MoveL RelTool (p1,5.500000,12.500000,6.000000,\Rx:=0.000000,\Ry:=0.000000),vel1,zoneval,Extruder\WObj:=Workobject_1;
MoveL RelTool (p1,3.000000,12.500000,6.000000,\Rx:=0.000000,\Ry:=0.000000),vel1,zoneval,Extruder\WObj:=Workobject_1;
MoveL RelTool (p1,5.000000,13.000000,6.000000,\Rx:=0.000000,\Ry:=-0.000000),vel1,zoneval,Extruder\WObj:=Workobject_1;
MoveL RelTool (p1,7.500000,13.000000,6.000000,\Rx:=0.000000,\Ry:=-0.000000),vel1,zoneval,Extruder\WObj:=Workobject_1;
MoveL RelTool (p1,10.000000,13.000000,6.000000,\Rx:=0.000000,\Ry:=-0.000000),vel1,zoneval,Extruder\WObj:=Workobject_1;
MoveL RelTool (p1,12.500000,13.000000,6.000000,\Rx:=0.000000,\Ry:=-0.000000),vel1,zoneval,Extruder\WObj:=Workobject_1;
MoveL RelTool (p1,15.000000,13.000000,6.000000,\Rx:=0.000000,\Ry:=-0.000000),vel1,zoneval,Extruder\WObj:=Workobject_1;
MoveL RelTool (p1,17.500000,13.000000,6.049338,\Rx:=0.000000,\Ry:=-1.971515),vel1,zoneval,Extruder\WObj:=Workobject_1;
MoveL RelTool (p1,20.000000,13.000000,6.980750,\Rx:=0.000000,\Ry:=-8.490094),vel1,zoneval,Extruder\WObj:=Workobject_1;
MoveL RelTool (p1,22.500000,13.000000,9.643620,\Rx:=0.000000,\Ry:=-9.749586),vel1,zoneval,Extruder\WObj:=Workobject_1;
MoveL RelTool (p1,25.000000,13.000000,11.616136,\Rx:=0.000000,\Ry:=-6.984613),vel1,zoneval,Extruder\WObj:=Workobject_1;
MoveL RelTool (p1,27.500000,13.000000,12.963548,\Rx:=0.000000,\Ry:=-5.267415),vel1,zoneval,Extruder\WObj:=Workobject_1;
MoveL RelTool (p1,30.000000,13.000000,13.961706,\Rx:=0.000000,\Ry:=-4.044321),vel1,zoneval,Extruder\WObj:=Workobject_1;
MoveL RelTool (p1,32.500000,13.000000,14.718653,\Rx:=0.000000,\Ry:=-3.050426),vel1,zoneval,Extruder\WObj:=Workobject_1;
MoveL RelTool (p1,35.000000,13.000000,15.272539,\Rx:=0.000000,\Ry:=-2.353997),vel1,zoneval,Extruder\WObj:=Workobject_1;
MoveL RelTool (p1,37.500000,13.000000,15.663580,\Rx:=0.000000,\Ry:=-1.455729),vel1,zoneval,Extruder\WObj:=Workobject_1;
MoveL RelTool (p1,40.000000,13.000000,15.887387,\Rx:=0.000000,\Ry:=-0.888959),vel1,zoneval,Extruder\WObj:=Workobject_1;
MoveL RelTool (p1,42.500000,13.000000,15.992154,\Rx:=0.000000,\Ry:=-0.087941),vel1,zoneval,Extruder\WObj:=Workobject_1;
MoveL RelTool (p1,45.000000,13.000000,15.941430,\Rx:=0.000000,\Ry:=0.668129),vel1,zoneval,Extruder\WObj:=Workobject_1;
MoveL RelTool (p1,47.500000,13.000000,15.759207,\Rx:=0.000000,\Ry:=1.496196),vel1,zoneval,Extruder\WObj:=Workobject_1;
MoveL RelTool (p1,50.000000,13.000000,15.420215,\Rx:=0.000000,\Ry:=2.179974),vel1,zoneval,Extruder\WObj:=Workobject_1;
MoveL RelTool (p1,52.500000,13.000000,14.925537,\Rx:=0.000000,\Ry:=3.343435),vel1,zoneval,Extruder\WObj:=Workobject_1;
MoveL RelTool (p1,55.000000,13.000000,14.234849,\Rx:=0.000000,\Ry:=3.932843),vel1,zoneval,Extruder\WObj:=Workobject_1;
MoveL RelTool (p1,57.500000,13.000000,13.324111,\Rx:=0.000000,\Ry:=5.119588),vel1,zoneval,Extruder\WObj:=Workobject_1;
MoveL RelTool (p1,60.000000,13.000000,12.115065,\Rx:=0.000000,\Ry:=6.738277),vel1,zoneval,Extruder\WObj:=Workobject_1;
MoveL RelTool (p1,62.500000,13.000000,10.412342,\Rx:=0.000000,\Ry:=9.301668),vel1,zoneval,Extruder\WObj:=Workobject_1;
MoveL RelTool (p1,65.000000,13.000000,7.669409,\Rx:=0.000000,\Ry:=9.245058),vel1,zoneval,Extruder\WObj:=Workobject_1;
MoveL RelTool (p1,67.500000,13.000000,6.209438,\Rx:=0.000000,\Ry:=3.081673),vel1,zoneval,Extruder\WObj:=Workobject_1;
MoveL RelTool (p1,70.000000,13.000000,6.000000,\Rx:=0.000000,\Ry:=-0.000000),vel1,zoneval,Extruder\WObj:=Workobject_1;
MoveL RelTool (p1,72.500000,13.000000,6.000000,\Rx:=0.000000,\Ry:=-0.000000),vel1,zoneval,Extruder\WObj:=Workobject_1;
MoveL RelTool (p1,75.000000,13.000000,6.000000,\Rx:=0.000000,\Ry:=-0.000000),vel1,zoneval,Extruder\WObj:=Workobject_1;
MoveL RelTool (p1,77.500000,13.000000,6.000000,\Rx:=0.000000,\Ry:=-0.000000),vel1,zoneval,Extruder\WObj:=Workobject_1;
MoveL RelTool (p1,80.000000,13.000000,6.000000,\Rx:=0.000000,\Ry:=-0.000000),vel1,zoneval,Extruder\WObj:=Workobject_1;
MoveL RelTool (p1,82.500000,13.000000,6.000000,\Rx:=0.000000,\Ry:=-0.000000),vel1,zoneval,Extruder\WObj:=Workobject_1;
MoveL RelTool (p1,80.500000,13.500000,6.000000,\Rx:=0.000000,\Ry:=0.000000),vel1,zoneval,Extruder\WObj:=Workobject_1;
MoveL RelTool (p1,78.000000,13.500000,6.000000,\Rx:=0.000000,\Ry:=0.000000),vel1,zoneval,Extruder\WObj:=Workobject_1;
MoveL RelTool (p1,75.500000,13.500000,6.000000,\Rx:=0.000000,\Ry:=0.000000),vel1,zoneval,Extruder\WObj:=Workobject_1;
MoveL RelTool (p1,73.000000,13.500000,6.000000,\Rx:=0.000000,\Ry:=0.000000),vel1,zoneval,Extruder\WObj:=Workobject_1;
MoveL RelTool (p1,70.500000,13.500000,6.000000,\Rx:=0.000000,\Ry:=0.000000),vel1,zoneval,Extruder\WObj:=Workobject_1;
MoveL RelTool (p1,68.000000,13.500000,6.086002,\Rx:=0.000000,\Ry:=3.081673),vel1,zoneval,Extruder\WObj:=Workobject_1;
MoveL RelTool (p1,65.500000,13.500000,7.225445,\Rx:=0.000000,\Ry:=9.245058),vel1,zoneval,Extruder\WObj:=Workobject_1;
MoveL RelTool (p1,63.000000,13.500000,9.965620,\Rx:=0.000000,\Ry:=9.278495),vel1,zoneval,Extruder\WObj:=Workobject_1;
MoveL RelTool (p1,60.500000,13.500000,11.822412,\Rx:=0.000000,\Ry:=6.739756),vel1,zoneval,Extruder\WObj:=Workobject_1;
MoveL RelTool (p1,58.000000,13.500000,13.112852,\Rx:=0.000000,\Ry:=5.083156),vel1,zoneval,Extruder\WObj:=Workobject_1;
MoveL RelTool (p1,55.500000,13.500000,14.075842,\Rx:=0.000000,\Ry:=3.914347),vel1,zoneval,Extruder\WObj:=Workobject_1;
MoveL RelTool (p1,53.000000,13.500000,14.791119,\Rx:=0.000000,\Ry:=3.343440),vel1,zoneval,Extruder\WObj:=Workobject_1;
MoveL RelTool (p1,50.500000,13.500000,15.333521,\Rx:=0.000000,\Ry:=2.179974),vel1,zoneval,Extruder\WObj:=Workobject_1;
MoveL RelTool (p1,48.000000,13.500000,15.700930,\Rx:=0.000000,\Ry:=1.469323),vel1,zoneval,Extruder\WObj:=Workobject_1;
MoveL RelTool (p1,45.500000,13.500000,15.915465,\Rx:=0.000000,\Ry:=0.668129),vel1,zoneval,Extruder\WObj:=Workobject_1;
MoveL RelTool (p1,43.000000,13.500000,15.995410,\Rx:=0.000000,\Ry:=-0.058203),vel1,zoneval,Extruder\WObj:=Workobject_1;
MoveL RelTool (p1,40.500000,13.500000,15.922527,\Rx:=0.000000,\Ry:=-0.858750),vel1,zoneval,Extruder\WObj:=Workobject_1;
MoveL RelTool (p1,38.000000,13.500000,15.720700,\Rx:=0.000000,\Ry:=-1.431827),vel1,zoneval,Extruder\WObj:=Workobject_1;
MoveL RelTool (p1,35.500000,13.500000,15.365736,\Rx:=0.000000,\Ry:=-2.353997),vel1,zoneval,Extruder\WObj:=Workobject_1;
MoveL RelTool (p1,33.000000,13.500000,14.841013,\Rx:=0.000000,\Ry:=-3.059013),vel1,zoneval,Extruder\WObj:=Workobject_1;
MoveL RelTool (p1,30.500000,13.500000,14.125926,\Rx:=0.000000,\Ry:=-4.044321),vel1,zoneval,Extruder\WObj:=Workobject_1;
MoveL RelTool (p1,28.000000,13.500000,13.182734,\Rx:=0.000000,\Ry:=-5.267415),vel1,zoneval,Extruder\WObj:=Workobject_1;
MoveL RelTool (p1,25.500000,13.500000,11.921360,\Rx:=0.000000,\Ry:=-6.957275),vel1,zoneval,Extruder\WObj:=Workobject_1;
MoveL RelTool (p1,23.000000,13.500000,10.124051,\Rx:=0.000000,\Ry:=-9.725837),vel1,zoneval,Extruder\WObj:=Workobject_1;
MoveL RelTool (p1,20.500000,13.500000,7.374287,\Rx:=0.000000,\Ry:=-8.490094),vel1,zoneval,Extruder\WObj:=Workobject_1;
MoveL RelTool (p1,18.000000,13.500000,6.127384,\Rx:=0.000000,\Ry:=-1.971515),vel1,zoneval,Extruder\WObj:=Workobject_1;
MoveL RelTool (p1,15.500000,13.500000,6.000000,\Rx:=0.000000,\Ry:=0.000000),vel1,zoneval,Extruder\WObj:=Workobject_1;
MoveL RelTool (p1,13.000000,13.500000,6.000000,\Rx:=0.000000,\Ry:=0.000000),vel1,zoneval,Extruder\WObj:=Workobject_1;
MoveL RelTool (p1,10.500000,13.500000,6.000000,\Rx:=0.000000,\Ry:=0.000000),vel1,zoneval,Extruder\WObj:=Workobject_1;
MoveL RelTool (p1,8.000000,13.500000,6.000000,\Rx:=0.000000,\Ry:=0.000000),vel1,zoneval,Extruder\WObj:=Workobject_1;
MoveL RelTool (p1,5.500000,13.500000,6.000000,\Rx:=0.000000,\Ry:=0.000000),vel1,zoneval,Extruder\WObj:=Workobject_1;
MoveL RelTool (p1,3.000000,13.500000,6.000000,\Rx:=0.000000,\Ry:=0.000000),vel1,zoneval,Extruder\WObj:=Workobject_1;
MoveL RelTool (p1,5.000000,14.000000,6.000000,\Rx:=0.000000,\Ry:=-0.000000),vel1,zoneval,Extruder\WObj:=Workobject_1;
MoveL RelTool (p1,7.500000,14.000000,6.000000,\Rx:=0.000000,\Ry:=-0.000000),vel1,zoneval,Extruder\WObj:=Workobject_1;
MoveL RelTool (p1,10.000000,14.000000,6.000000,\Rx:=0.000000,\Ry:=-0.000000),vel1,zoneval,Extruder\WObj:=Workobject_1;
MoveL RelTool (p1,12.500000,14.000000,6.000000,\Rx:=0.000000,\Ry:=-0.000000),vel1,zoneval,Extruder\WObj:=Workobject_1;
MoveL RelTool (p1,15.000000,14.000000,6.000000,\Rx:=0.000000,\Ry:=-0.000000),vel1,zoneval,Extruder\WObj:=Workobject_1;
MoveL RelTool (p1,17.500000,14.000000,6.049338,\Rx:=0.000000,\Ry:=-1.971515),vel1,zoneval,Extruder\WObj:=Workobject_1;
MoveL RelTool (p1,20.000000,14.000000,6.980750,\Rx:=0.000000,\Ry:=-8.490094),vel1,zoneval,Extruder\WObj:=Workobject_1;
MoveL RelTool (p1,22.500000,14.000000,9.646646,\Rx:=0.000000,\Ry:=-9.702002),vel1,zoneval,Extruder\WObj:=Workobject_1;
MoveL RelTool (p1,25.000000,14.000000,11.618390,\Rx:=0.000000,\Ry:=-6.929866),vel1,zoneval,Extruder\WObj:=Workobject_1;
MoveL RelTool (p1,27.500000,14.000000,12.962881,\Rx:=0.000000,\Ry:=-5.267415),vel1,zoneval,Extruder\WObj:=Workobject_1;
MoveL RelTool (p1,30.000000,14.000000,13.961372,\Rx:=0.000000,\Ry:=-4.044321),vel1,zoneval,Extruder\WObj:=Workobject_1;
MoveL RelTool (p1,32.500000,14.000000,14.718387,\Rx:=0.000000,\Ry:=-3.067598),vel1,zoneval,Extruder\WObj:=Workobject_1;
MoveL RelTool (p1,35.000000,14.000000,15.271916,\Rx:=0.000000,\Ry:=-2.353997),vel1,zoneval,Extruder\WObj:=Workobject_1;
MoveL RelTool (p1,37.500000,14.000000,15.664889,\Rx:=0.000000,\Ry:=-1.407915),vel1,zoneval,Extruder\WObj:=Workobject_1;
MoveL RelTool (p1,40.000000,14.000000,15.890119,\Rx:=0.000000,\Ry:=-0.828532),vel1,zoneval,Extruder\WObj:=Workobject_1;
MoveL RelTool (p1,42.500000,14.000000,15.994096,\Rx:=0.000000,\Ry:=-0.028464),vel1,zoneval,Extruder\WObj:=Workobject_1;
MoveL RelTool (p1,45.000000,14.000000,15.942022,\Rx:=0.000000,\Ry:=0.668129),vel1,zoneval,Extruder\WObj:=Workobject_1;
MoveL RelTool (p1,47.500000,14.000000,15.758568,\Rx:=0.000000,\Ry:=1.442437),vel1,zoneval,Extruder\WObj:=Workobject_1;
MoveL RelTool (p1,50.000000,14.000000,15.419734,\Rx:=0.000000,\Ry:=2.179974),vel1,zoneval,Extruder\WObj:=Workobject_1;
MoveL RelTool (p1,52.500000,14.000000,14.925501,\Rx:=0.000000,\Ry:=3.287338),vel1,zoneval,Extruder\WObj:=Workobject_1;
MoveL RelTool (p1,55.000000,14.000000,14.234333,\Rx:=0.000000,\Ry:=3.895833),vel1,zoneval,Extruder\WObj:=Workobject_1;
MoveL RelTool (p1,57.500000,14.000000,13.323479,\Rx:=0.000000,\Ry:=5.046636),vel1,zoneval,Extruder\WObj:=Workobject_1;
MoveL RelTool (p1,60.000000,14.000000,12.114788,\Rx:=0.000000,\Ry:=6.741235),vel1,zoneval,Extruder\WObj:=Workobject_1;
MoveL RelTool (p1,62.500000,14.000000,10.411534,\Rx:=0.000000,\Ry:=9.255247),vel1,zoneval,Extruder\WObj:=Workobject_1;
MoveL RelTool (p1,65.000000,14.000000,7.669409,\Rx:=0.000000,\Ry:=9.245058),vel1,zoneval,Extruder\WObj:=Workobject_1;
MoveL RelTool (p1,67.500000,14.000000,6.209438,\Rx:=0.000000,\Ry:=3.081673),vel1,zoneval,Extruder\WObj:=Workobject_1;
MoveL RelTool (p1,70.000000,14.000000,6.000000,\Rx:=0.000000,\Ry:=-0.000000),vel1,zoneval,Extruder\WObj:=Workobject_1;
MoveL RelTool (p1,72.500000,14.000000,6.000000,\Rx:=0.000000,\Ry:=-0.000000),vel1,zoneval,Extruder\WObj:=Workobject_1;
MoveL RelTool (p1,75.000000,14.000000,6.000000,\Rx:=0.000000,\Ry:=-0.000000),vel1,zoneval,Extruder\WObj:=Workobject_1;
MoveL RelTool (p1,77.500000,14.000000,6.000000,\Rx:=0.000000,\Ry:=-0.000000),vel1,zoneval,Extruder\WObj:=Workobject_1;
MoveL RelTool (p1,80.000000,14.000000,6.000000,\Rx:=0.000000,\Ry:=-0.000000),vel1,zoneval,Extruder\WObj:=Workobject_1;
MoveL RelTool (p1,82.500000,14.000000,6.000000,\Rx:=0.000000,\Ry:=-0.000000),vel1,zoneval,Extruder\WObj:=Workobject_1;
MoveL RelTool (p1,80.500000,14.500000,6.000000,\Rx:=0.000000,\Ry:=0.000000),vel1,zoneval,Extruder\WObj:=Workobject_1;
MoveL RelTool (p1,78.000000,14.500000,6.000000,\Rx:=0.000000,\Ry:=0.000000),vel1,zoneval,Extruder\WObj:=Workobject_1;
MoveL RelTool (p1,75.500000,14.500000,6.000000,\Rx:=0.000000,\Ry:=0.000000),vel1,zoneval,Extruder\WObj:=Workobject_1;
MoveL RelTool (p1,73.000000,14.500000,6.000000,\Rx:=0.000000,\Ry:=0.000000),vel1,zoneval,Extruder\WObj:=Workobject_1;
MoveL RelTool (p1,70.500000,14.500000,6.000000,\Rx:=0.000000,\Ry:=0.000000),vel1,zoneval,Extruder\WObj:=Workobject_1;
MoveL RelTool (p1,68.000000,14.500000,6.086002,\Rx:=0.000000,\Ry:=3.081673),vel1,zoneval,Extruder\WObj:=Workobject_1;
MoveL RelTool (p1,65.500000,14.500000,7.225445,\Rx:=0.000000,\Ry:=9.245058),vel1,zoneval,Extruder\WObj:=Workobject_1;
MoveL RelTool (p1,63.000000,14.500000,9.968088,\Rx:=0.000000,\Ry:=9.231924),vel1,zoneval,Extruder\WObj:=Workobject_1;
MoveL RelTool (p1,60.500000,14.500000,11.821979,\Rx:=0.000000,\Ry:=6.742713),vel1,zoneval,Extruder\WObj:=Workobject_1;
MoveL RelTool (p1,58.000000,14.500000,13.115420,\Rx:=0.000000,\Ry:=5.013820),vel1,zoneval,Extruder\WObj:=Workobject_1;
MoveL RelTool (p1,55.500000,14.500000,14.076926,\Rx:=0.000000,\Ry:=3.877303),vel1,zoneval,Extruder\WObj:=Workobject_1;
MoveL RelTool (p1,53.000000,14.500000,14.795076,\Rx:=0.000000,\Ry:=3.248438),vel1,zoneval,Extruder\WObj:=Workobject_1;
MoveL RelTool (p1,50.500000,14.500000,15.333041,\Rx:=0.000000,\Ry:=2.179974),vel1,zoneval,Extruder\WObj:=Workobject_1;
MoveL RelTool (p1,48.000000,14.500000,15.702430,\Rx:=0.000000,\Ry:=1.415537),vel1,zoneval,Extruder\WObj:=Workobject_1;
MoveL RelTool (p1,45.500000,14.500000,15.916057,\Rx:=0.000000,\Ry:=0.668129),vel1,zoneval,Extruder\WObj:=Workobject_1;
MoveL RelTool (p1,43.000000,14.500000,15.995016,\Rx:=0.000000,\Ry:=0.001275),vel1,zoneval,Extruder\WObj:=Workobject_1;
MoveL RelTool (p1,40.500000,14.500000,15.923861,\Rx:=0.000000,\Ry:=-0.823311),vel1,zoneval,Extruder\WObj:=Workobject_1;
MoveL RelTool (p1,38.000000,14.500000,15.720108,\Rx:=0.000000,\Ry:=-1.383993),vel1,zoneval,Extruder\WObj:=Workobject_1;
MoveL RelTool (p1,35.500000,14.500000,15.365113,\Rx:=0.000000,\Ry:=-2.353997),vel1,zoneval,Extruder\WObj:=Workobject_1;
MoveL RelTool (p1,33.000000,14.500000,14.841462,\Rx:=0.000000,\Ry:=-3.076179),vel1,zoneval,Extruder\WObj:=Workobject_1;
MoveL RelTool (p1,30.500000,14.500000,14.125592,\Rx:=0.000000,\Ry:=-4.044321),vel1,zoneval,Extruder\WObj:=Workobject_1;
MoveL RelTool (p1,28.000000,14.500000,13.182067,\Rx:=0.000000,\Ry:=-5.267415),vel1,zoneval,Extruder\WObj:=Workobject_1;
MoveL RelTool (p1,25.500000,14.500000,11.920669,\Rx:=0.000000,\Ry:=-6.904626),vel1,zoneval,Extruder\WObj:=Workobject_1;
MoveL RelTool (p1,23.000000,14.500000,10.123494,\Rx:=0.000000,\Ry:=-9.678082),vel1,zoneval,Extruder\WObj:=Workobject_1;
MoveL RelTool (p1,20.500000,14.500000,7.374287,\Rx:=0.000000,\Ry:=-8.490094),vel1,zoneval,Extruder\WObj:=Workobject_1;
MoveL RelTool (p1,18.000000,14.500000,6.127384,\Rx:=0.000000,\Ry:=-1.971515),vel1,zoneval,Extruder\WObj:=Workobject_1;
MoveL RelTool (p1,15.500000,14.500000,6.000000,\Rx:=0.000000,\Ry:=0.000000),vel1,zoneval,Extruder\WObj:=Workobject_1;
MoveL RelTool (p1,13.000000,14.500000,6.000000,\Rx:=0.000000,\Ry:=0.000000),vel1,zoneval,Extruder\WObj:=Workobject_1;
MoveL RelTool (p1,10.500000,14.500000,6.000000,\Rx:=0.000000,\Ry:=0.000000),vel1,zoneval,Extruder\WObj:=Workobject_1;
MoveL RelTool (p1,8.000000,14.500000,6.000000,\Rx:=0.000000,\Ry:=0.000000),vel1,zoneval,Extruder\WObj:=Workobject_1;
MoveL RelTool (p1,5.500000,14.500000,6.000000,\Rx:=0.000000,\Ry:=0.000000),vel1,zoneval,Extruder\WObj:=Workobject_1;
MoveL RelTool (p1,3.000000,14.500000,6.000000,\Rx:=0.000000,\Ry:=0.000000),vel1,zoneval,Extruder\WObj:=Workobject_1;
MoveL RelTool (p1,5.000000,15.000000,6.000000,\Rx:=0.000000,\Ry:=-0.000000),vel1,zoneval,Extruder\WObj:=Workobject_1;
MoveL RelTool (p1,7.500000,15.000000,6.000000,\Rx:=0.000000,\Ry:=-0.000000),vel1,zoneval,Extruder\WObj:=Workobject_1;
MoveL RelTool (p1,10.000000,15.000000,6.000000,\Rx:=0.000000,\Ry:=-0.000000),vel1,zoneval,Extruder\WObj:=Workobject_1;
MoveL RelTool (p1,12.500000,15.000000,6.000000,\Rx:=0.000000,\Ry:=-0.000000),vel1,zoneval,Extruder\WObj:=Workobject_1;
MoveL RelTool (p1,15.000000,15.000000,6.000000,\Rx:=0.000000,\Ry:=-0.000000),vel1,zoneval,Extruder\WObj:=Workobject_1;
MoveL RelTool (p1,17.500000,15.000000,6.049338,\Rx:=0.000000,\Ry:=-1.971515),vel1,zoneval,Extruder\WObj:=Workobject_1;
MoveL RelTool (p1,20.000000,15.000000,6.980750,\Rx:=0.000000,\Ry:=-8.490094),vel1,zoneval,Extruder\WObj:=Workobject_1;
MoveL RelTool (p1,22.500000,15.000000,9.649672,\Rx:=0.000000,\Ry:=-9.654076),vel1,zoneval,Extruder\WObj:=Workobject_1;
MoveL RelTool (p1,25.000000,15.000000,11.619515,\Rx:=0.000000,\Ry:=-6.895951),vel1,zoneval,Extruder\WObj:=Workobject_1;
MoveL RelTool (p1,27.500000,15.000000,12.962213,\Rx:=0.000000,\Ry:=-5.267415),vel1,zoneval,Extruder\WObj:=Workobject_1;
MoveL RelTool (p1,30.000000,15.000000,13.961039,\Rx:=0.000000,\Ry:=-4.044321),vel1,zoneval,Extruder\WObj:=Workobject_1;
MoveL RelTool (p1,32.500000,15.000000,14.718121,\Rx:=0.000000,\Ry:=-3.084758),vel1,zoneval,Extruder\WObj:=Workobject_1;
MoveL RelTool (p1,35.000000,15.000000,15.271293,\Rx:=0.000000,\Ry:=-2.353997),vel1,zoneval,Extruder\WObj:=Workobject_1;
MoveL RelTool (p1,37.500000,15.000000,15.666198,\Rx:=0.000000,\Ry:=-1.360061),vel1,zoneval,Extruder\WObj:=Workobject_1;
MoveL RelTool (p1,40.000000,15.000000,15.892850,\Rx:=0.000000,\Ry:=-0.823311),vel1,zoneval,Extruder\WObj:=Workobject_1;
MoveL RelTool (p1,42.500000,15.000000,15.995638,\Rx:=0.000000,\Ry:=0.020861),vel1,zoneval,Extruder\WObj:=Workobject_1;
MoveL RelTool (p1,45.000000,15.000000,15.942614,\Rx:=0.000000,\Ry:=0.668129),vel1,zoneval,Extruder\WObj:=Workobject_1;
MoveL RelTool (p1,47.500000,15.000000,15.757929,\Rx:=0.000000,\Ry:=1.392190),vel1,zoneval,Extruder\WObj:=Workobject_1;
MoveL RelTool (p1,50.000000,15.000000,15.419254,\Rx:=0.000000,\Ry:=2.179974),vel1,zoneval,Extruder\WObj:=Workobject_1;
MoveL RelTool (p1,52.500000,15.000000,14.925466,\Rx:=0.000000,\Ry:=3.209475),vel1,zoneval,Extruder\WObj:=Workobject_1;
MoveL RelTool (p1,55.000000,15.000000,14.233818,\Rx:=0.000000,\Ry:=3.858755),vel1,zoneval,Extruder\WObj:=Workobject_1;
MoveL RelTool (p1,57.500000,15.000000,13.322847,\Rx:=0.000000,\Ry:=5.013820),vel1,zoneval,Extruder\WObj:=Workobject_1;
MoveL RelTool (p1,60.000000,15.000000,12.114512,\Rx:=0.000000,\Ry:=6.744192),vel1,zoneval,Extruder\WObj:=Workobject_1;
MoveL RelTool (p1,62.500000,15.000000,10.410726,\Rx:=0.000000,\Ry:=9.208524),vel1,zoneval,Extruder\WObj:=Workobject_1;
MoveL RelTool (p1,65.000000,15.000000,7.669409,\Rx:=0.000000,\Ry:=9.245058),vel1,zoneval,Extruder\WObj:=Workobject_1;
MoveL RelTool (p1,67.500000,15.000000,6.209438,\Rx:=0.000000,\Ry:=3.081673),vel1,zoneval,Extruder\WObj:=Workobject_1;
MoveL RelTool (p1,70.000000,15.000000,6.000000,\Rx:=0.000000,\Ry:=-0.000000),vel1,zoneval,Extruder\WObj:=Workobject_1;
MoveL RelTool (p1,72.500000,15.000000,6.000000,\Rx:=0.000000,\Ry:=-0.000000),vel1,zoneval,Extruder\WObj:=Workobject_1;
MoveL RelTool (p1,75.000000,15.000000,6.000000,\Rx:=0.000000,\Ry:=-0.000000),vel1,zoneval,Extruder\WObj:=Workobject_1;
MoveL RelTool (p1,77.500000,15.000000,6.000000,\Rx:=0.000000,\Ry:=-0.000000),vel1,zoneval,Extruder\WObj:=Workobject_1;
MoveL RelTool (p1,80.000000,15.000000,6.000000,\Rx:=0.000000,\Ry:=-0.000000),vel1,zoneval,Extruder\WObj:=Workobject_1;
MoveL RelTool (p1,82.500000,15.000000,6.000000,\Rx:=0.000000,\Ry:=-0.000000),vel1,zoneval,Extruder\WObj:=Workobject_1;
MoveL RelTool (p1,80.500000,15.500000,6.000000,\Rx:=0.000000,\Ry:=0.000000),vel1,zoneval,Extruder\WObj:=Workobject_1;
MoveL RelTool (p1,78.000000,15.500000,6.000000,\Rx:=0.000000,\Ry:=0.000000),vel1,zoneval,Extruder\WObj:=Workobject_1;
MoveL RelTool (p1,75.500000,15.500000,6.000000,\Rx:=0.000000,\Ry:=0.000000),vel1,zoneval,Extruder\WObj:=Workobject_1;
MoveL RelTool (p1,73.000000,15.500000,6.000000,\Rx:=0.000000,\Ry:=0.000000),vel1,zoneval,Extruder\WObj:=Workobject_1;
MoveL RelTool (p1,70.500000,15.500000,6.000000,\Rx:=0.000000,\Ry:=0.000000),vel1,zoneval,Extruder\WObj:=Workobject_1;
MoveL RelTool (p1,68.000000,15.500000,6.086002,\Rx:=0.000000,\Ry:=3.081673),vel1,zoneval,Extruder\WObj:=Workobject_1;
MoveL RelTool (p1,65.500000,15.500000,7.225445,\Rx:=0.000000,\Ry:=9.245058),vel1,zoneval,Extruder\WObj:=Workobject_1;
MoveL RelTool (p1,63.000000,15.500000,9.970555,\Rx:=0.000000,\Ry:=9.185048),vel1,zoneval,Extruder\WObj:=Workobject_1;
MoveL RelTool (p1,60.500000,15.500000,11.821547,\Rx:=0.000000,\Ry:=6.745670),vel1,zoneval,Extruder\WObj:=Workobject_1;
MoveL RelTool (p1,58.000000,15.500000,13.114788,\Rx:=0.000000,\Ry:=5.013820),vel1,zoneval,Extruder\WObj:=Workobject_1;
MoveL RelTool (p1,55.500000,15.500000,14.078010,\Rx:=0.000000,\Ry:=3.840191),vel1,zoneval,Extruder\WObj:=Workobject_1;
MoveL RelTool (p1,53.000000,15.500000,14.798306,\Rx:=0.000000,\Ry:=3.170451),vel1,zoneval,Extruder\WObj:=Workobject_1;
MoveL RelTool (p1,50.500000,15.500000,15.332561,\Rx:=0.000000,\Ry:=2.179974),vel1,zoneval,Extruder\WObj:=Workobject_1;
MoveL RelTool (p1,48.000000,15.500000,15.703432,\Rx:=0.000000,\Ry:=1.374237),vel1,zoneval,Extruder\WObj:=Workobject_1;
MoveL RelTool (p1,45.500000,15.500000,15.916648,\Rx:=0.000000,\Ry:=0.668129),vel1,zoneval,Extruder\WObj:=Workobject_1;
MoveL RelTool (p1,43.000000,15.500000,15.994622,\Rx:=0.000000,\Ry:=0.023524),vel1,zoneval,Extruder\WObj:=Workobject_1;
MoveL RelTool (p1,40.500000,15.500000,15.926593,\Rx:=0.000000,\Ry:=-0.823311),vel1,zoneval,Extruder\WObj:=Workobject_1;
MoveL RelTool (p1,38.000000,15.500000,15.719515,\Rx:=0.000000,\Ry:=-1.336120),vel1,zoneval,Extruder\WObj:=Workobject_1;
MoveL RelTool (p1,35.500000,15.500000,15.364490,\Rx:=0.000000,\Ry:=-2.353997),vel1,zoneval,Extruder\WObj:=Workobject_1;
MoveL RelTool (p1,33.000000,15.500000,14.841911,\Rx:=0.000000,\Ry:=-3.093334),vel1,zoneval,Extruder\WObj:=Workobject_1;
MoveL RelTool (p1,30.500000,15.500000,14.125258,\Rx:=0.000000,\Ry:=-4.044321),vel1,zoneval,Extruder\WObj:=Workobject_1;
MoveL RelTool (p1,28.000000,15.500000,13.181399,\Rx:=0.000000,\Ry:=-5.267415),vel1,zoneval,Extruder\WObj:=Workobject_1;
MoveL RelTool (p1,25.500000,15.500000,11.919977,\Rx:=0.000000,\Ry:=-6.887269),vel1,zoneval,Extruder\WObj:=Workobject_1;
MoveL RelTool (p1,23.000000,15.500000,10.122937,\Rx:=0.000000,\Ry:=-9.629984),vel1,zoneval,Extruder\WObj:=Workobject_1;
MoveL RelTool (p1,20.500000,15.500000,7.374287,\Rx:=0.000000,\Ry:=-8.490094),vel1,zoneval,Extruder\WObj:=Workobject_1;
MoveL RelTool (p1,18.000000,15.500000,6.127384,\Rx:=0.000000,\Ry:=-1.971515),vel1,zoneval,Extruder\WObj:=Workobject_1;
MoveL RelTool (p1,15.500000,15.500000,6.000000,\Rx:=0.000000,\Ry:=0.000000),vel1,zoneval,Extruder\WObj:=Workobject_1;
MoveL RelTool (p1,13.000000,15.500000,6.000000,\Rx:=0.000000,\Ry:=0.000000),vel1,zoneval,Extruder\WObj:=Workobject_1;
MoveL RelTool (p1,10.500000,15.500000,6.000000,\Rx:=0.000000,\Ry:=0.000000),vel1,zoneval,Extruder\WObj:=Workobject_1;
MoveL RelTool (p1,8.000000,15.500000,6.000000,\Rx:=0.000000,\Ry:=0.000000),vel1,zoneval,Extruder\WObj:=Workobject_1;
MoveL RelTool (p1,5.500000,15.500000,6.000000,\Rx:=0.000000,\Ry:=0.000000),vel1,zoneval,Extruder\WObj:=Workobject_1;
MoveL RelTool (p1,3.000000,15.500000,6.000000,\Rx:=0.000000,\Ry:=0.000000),vel1,zoneval,Extruder\WObj:=Workobject_1;
MoveL RelTool (p1,5.000000,16.000000,6.000000,\Rx:=0.000000,\Ry:=-0.000000),vel1,zoneval,Extruder\WObj:=Workobject_1;
MoveL RelTool (p1,7.500000,16.000000,6.000000,\Rx:=0.000000,\Ry:=-0.000000),vel1,zoneval,Extruder\WObj:=Workobject_1;
MoveL RelTool (p1,10.000000,16.000000,6.000000,\Rx:=0.000000,\Ry:=-0.000000),vel1,zoneval,Extruder\WObj:=Workobject_1;
MoveL RelTool (p1,12.500000,16.000000,6.000000,\Rx:=0.000000,\Ry:=-0.000000),vel1,zoneval,Extruder\WObj:=Workobject_1;
MoveL RelTool (p1,15.000000,16.000000,6.000000,\Rx:=0.000000,\Ry:=-0.000000),vel1,zoneval,Extruder\WObj:=Workobject_1;
MoveL RelTool (p1,17.500000,16.000000,6.049338,\Rx:=0.000000,\Ry:=-1.971515),vel1,zoneval,Extruder\WObj:=Workobject_1;
MoveL RelTool (p1,20.000000,16.000000,6.980750,\Rx:=0.000000,\Ry:=-8.490094),vel1,zoneval,Extruder\WObj:=Workobject_1;
MoveL RelTool (p1,22.500000,16.000000,9.652698,\Rx:=0.000000,\Ry:=-9.605805),vel1,zoneval,Extruder\WObj:=Workobject_1;
MoveL RelTool (p1,25.000000,16.000000,11.619752,\Rx:=0.000000,\Ry:=-6.878580),vel1,zoneval,Extruder\WObj:=Workobject_1;
MoveL RelTool (p1,27.500000,16.000000,12.961545,\Rx:=0.000000,\Ry:=-5.267415),vel1,zoneval,Extruder\WObj:=Workobject_1;
MoveL RelTool (p1,30.000000,16.000000,13.960705,\Rx:=0.000000,\Ry:=-4.044321),vel1,zoneval,Extruder\WObj:=Workobject_1;
MoveL RelTool (p1,32.500000,16.000000,14.717855,\Rx:=0.000000,\Ry:=-3.101906),vel1,zoneval,Extruder\WObj:=Workobject_1;
MoveL RelTool (p1,35.000000,16.000000,15.270669,\Rx:=0.000000,\Ry:=-2.353997),vel1,zoneval,Extruder\WObj:=Workobject_1;
MoveL RelTool (p1,37.500000,16.000000,15.667148,\Rx:=0.000000,\Ry:=-1.321199),vel1,zoneval,Extruder\WObj:=Workobject_1;
MoveL RelTool (p1,40.000000,16.000000,15.895582,\Rx:=0.000000,\Ry:=-0.823311),vel1,zoneval,Extruder\WObj:=Workobject_1;
MoveL RelTool (p1,42.500000,16.000000,15.995453,\Rx:=0.000000,\Ry:=0.026186),vel1,zoneval,Extruder\WObj:=Workobject_1;
MoveL RelTool (p1,45.000000,16.000000,15.943206,\Rx:=0.000000,\Ry:=0.668129),vel1,zoneval,Extruder\WObj:=Workobject_1;
MoveL RelTool (p1,47.500000,16.000000,15.757289,\Rx:=0.000000,\Ry:=1.356278),vel1,zoneval,Extruder\WObj:=Workobject_1;
MoveL RelTool (p1,50.000000,16.000000,15.418774,\Rx:=0.000000,\Ry:=2.179974),vel1,zoneval,Extruder\WObj:=Workobject_1;
MoveL RelTool (p1,52.500000,16.000000,14.925430,\Rx:=0.000000,\Ry:=3.131366),vel1,zoneval,Extruder\WObj:=Workobject_1;
MoveL RelTool (p1,55.000000,16.000000,14.233302,\Rx:=0.000000,\Ry:=3.821610),vel1,zoneval,Extruder\WObj:=Workobject_1;
MoveL RelTool (p1,57.500000,16.000000,13.322215,\Rx:=0.000000,\Ry:=5.013820),vel1,zoneval,Extruder\WObj:=Workobject_1;
MoveL RelTool (p1,60.000000,16.000000,12.114235,\Rx:=0.000000,\Ry:=6.747148),vel1,zoneval,Extruder\WObj:=Workobject_1;
MoveL RelTool (p1,62.500000,16.000000,10.409918,\Rx:=0.000000,\Ry:=9.161496),vel1,zoneval,Extruder\WObj:=Workobject_1;
MoveL RelTool (p1,65.000000,16.000000,7.669409,\Rx:=0.000000,\Ry:=9.245058),vel1,zoneval,Extruder\WObj:=Workobject_1;
MoveL RelTool (p1,67.500000,16.000000,6.209438,\Rx:=0.000000,\Ry:=3.081673),vel1,zoneval,Extruder\WObj:=Workobject_1;
MoveL RelTool (p1,70.000000,16.000000,6.000000,\Rx:=0.000000,\Ry:=-0.000000),vel1,zoneval,Extruder\WObj:=Workobject_1;
MoveL RelTool (p1,72.500000,16.000000,6.000000,\Rx:=0.000000,\Ry:=-0.000000),vel1,zoneval,Extruder\WObj:=Workobject_1;
MoveL RelTool (p1,75.000000,16.000000,6.000000,\Rx:=0.000000,\Ry:=-0.000000),vel1,zoneval,Extruder\WObj:=Workobject_1;
MoveL RelTool (p1,77.500000,16.000000,6.000000,\Rx:=0.000000,\Ry:=-0.000000),vel1,zoneval,Extruder\WObj:=Workobject_1;
MoveL RelTool (p1,80.000000,16.000000,6.000000,\Rx:=0.000000,\Ry:=-0.000000),vel1,zoneval,Extruder\WObj:=Workobject_1;
MoveL RelTool (p1,82.500000,16.000000,6.000000,\Rx:=0.000000,\Ry:=-0.000000),vel1,zoneval,Extruder\WObj:=Workobject_1;



MoveL RelTool (p1,82.500000,16.000000,70.000000,\Rx:=0.000000,\Ry:=-0.000000),vel1,zoneval,Extruder\WObj:=Workobject_1;



MoveL RelTool (p1,3.000000,3.000000,70.000000,\Rx:=0.000000,\Ry:=-0.000000),vel1,zoneval,Extruder\WObj:=Workobject_1;




MoveL RelTool (p1,3.000000,3.000000,6.500000,\Rx:=0.000000,\Ry:=0.000000),vel1,z0,Extruder\WObj:=Workobject_1;
MoveL RelTool (p1,16.889791,3.000000,6.500000,\Rx:=0.000000,\Ry:=0.000000),vel1,z0,Extruder\WObj:=Workobject_1;
MoveL RelTool (p1,17.693081,3.000000,6.564949,\Rx:=0.000000,\Ry:=0.000000),vel1,z0,Extruder\WObj:=Workobject_1;
MoveL RelTool (p1,18.475496,3.000000,6.758109,\Rx:=0.000000,\Ry:=0.000000),vel1,z0,Extruder\WObj:=Workobject_1;
MoveL RelTool (p1,19.216721,3.000000,7.074461,\Rx:=0.000000,\Ry:=0.000000),vel1,z0,Extruder\WObj:=Workobject_1;
MoveL RelTool (p1,19.897491,3.000000,7.505786,\Rx:=0.000000,\Ry:=0.000000),vel1,z0,Extruder\WObj:=Workobject_1;
MoveL RelTool (p1,20.500122,3.000000,8.040880,\Rx:=0.000000,\Ry:=0.000000),vel1,z0,Extruder\WObj:=Workobject_1;
MoveL RelTool (p1,21.008959,3.000000,8.665841,\Rx:=0.000000,\Ry:=0.000000),vel1,z0,Extruder\WObj:=Workobject_1;
MoveL RelTool (p1,21.655001,3.000000,9.492284,\Rx:=0.000000,\Ry:=0.000000),vel1,z0,Extruder\WObj:=Workobject_1;
MoveL RelTool (p1,22.745361,3.000000,10.576250,\Rx:=0.000000,\Ry:=0.000000),vel1,z0,Extruder\WObj:=Workobject_1;
MoveL RelTool (p1,24.141754,3.000000,11.657135,\Rx:=0.000000,\Ry:=0.000000),vel1,z0,Extruder\WObj:=Workobject_1;
MoveL RelTool (p1,25.864042,3.000000,12.709541,\Rx:=0.000000,\Ry:=0.000000),vel1,z0,Extruder\WObj:=Workobject_1;
MoveL RelTool (p1,27.915775,3.000000,13.697697,\Rx:=0.000000,\Ry:=0.000000),vel1,z0,Extruder\WObj:=Workobject_1;
MoveL RelTool (p1,30.224897,3.000000,14.569467,\Rx:=0.000000,\Ry:=0.000000),vel1,z0,Extruder\WObj:=Workobject_1;
MoveL RelTool (p1,32.769985,3.000000,15.305704,\Rx:=0.000000,\Ry:=0.000000),vel1,z0,Extruder\WObj:=Workobject_1;
MoveL RelTool (p1,35.546967,3.000000,15.885172,\Rx:=0.000000,\Ry:=0.000000),vel1,z0,Extruder\WObj:=Workobject_1;
MoveL RelTool (p1,38.467556,3.000000,16.278698,\Rx:=0.000000,\Ry:=0.000000),vel1,z0,Extruder\WObj:=Workobject_1;
MoveL RelTool (p1,41.456455,3.000000,16.476196,\Rx:=0.000000,\Ry:=0.000000),vel1,z0,Extruder\WObj:=Workobject_1;
MoveL RelTool (p1,44.466969,3.000000,16.473138,\Rx:=0.000000,\Ry:=0.000000),vel1,z0,Extruder\WObj:=Workobject_1;
MoveL RelTool (p1,47.447681,3.000000,16.270333,\Rx:=0.000000,\Ry:=0.000000),vel1,z0,Extruder\WObj:=Workobject_1;
MoveL RelTool (p1,50.292072,3.000000,15.884033,\Rx:=0.000000,\Ry:=0.000000),vel1,z0,Extruder\WObj:=Workobject_1;
MoveL RelTool (p1,52.986897,3.000000,15.324379,\Rx:=0.000000,\Ry:=0.000000),vel1,z0,Extruder\WObj:=Workobject_1;
MoveL RelTool (p1,55.503719,3.000000,14.603756,\Rx:=0.000000,\Ry:=0.000000),vel1,z0,Extruder\WObj:=Workobject_1;
MoveL RelTool (p1,57.756004,3.000000,13.765661,\Rx:=0.000000,\Ry:=0.000000),vel1,z0,Extruder\WObj:=Workobject_1;
MoveL RelTool (p1,59.724201,3.000000,12.840277,\Rx:=0.000000,\Ry:=0.000000),vel1,z0,Extruder\WObj:=Workobject_1;
MoveL RelTool (p1,61.421394,3.000000,11.838728,\Rx:=0.000000,\Ry:=0.000000),vel1,z0,Extruder\WObj:=Workobject_1;
MoveL RelTool (p1,62.837132,3.000000,10.789865,\Rx:=0.000000,\Ry:=0.000000),vel1,z0,Extruder\WObj:=Workobject_1;
MoveL RelTool (p1,63.967651,3.000000,9.724504,\Rx:=0.000000,\Ry:=0.000000),vel1,z0,Extruder\WObj:=Workobject_1;
MoveL RelTool (p1,64.823410,3.000000,8.665841,\Rx:=0.000000,\Ry:=0.000000),vel1,z0,Extruder\WObj:=Workobject_1;
MoveL RelTool (p1,65.332253,3.000000,8.040880,\Rx:=0.000000,\Ry:=0.000000),vel1,z0,Extruder\WObj:=Workobject_1;
MoveL RelTool (p1,65.934883,3.000000,7.505786,\Rx:=0.000000,\Ry:=0.000000),vel1,z0,Extruder\WObj:=Workobject_1;
MoveL RelTool (p1,66.615646,3.000000,7.074461,\Rx:=0.000000,\Ry:=0.000000),vel1,z0,Extruder\WObj:=Workobject_1;
MoveL RelTool (p1,67.356880,3.000000,6.758109,\Rx:=0.000000,\Ry:=0.000000),vel1,z0,Extruder\WObj:=Workobject_1;
MoveL RelTool (p1,68.139290,3.000000,6.564949,\Rx:=0.000000,\Ry:=0.000000),vel1,z0,Extruder\WObj:=Workobject_1;
MoveL RelTool (p1,68.942581,3.000000,6.500000,\Rx:=0.000000,\Ry:=0.000000),vel1,z0,Extruder\WObj:=Workobject_1;
MoveL RelTool (p1,82.832375,3.000000,6.500000,\Rx:=0.000000,\Ry:=0.000000),vel1,z0,Extruder\WObj:=Workobject_1;
MoveL RelTool (p1,82.832375,16.000000,6.500000,\Rx:=0.000000,\Ry:=0.000000),vel1,z0,Extruder\WObj:=Workobject_1;
MoveL RelTool (p1,68.942581,16.000000,6.500000,\Rx:=0.000000,\Ry:=0.000000),vel1,z0,Extruder\WObj:=Workobject_1;
MoveL RelTool (p1,68.139290,16.000000,6.564949,\Rx:=0.000000,\Ry:=0.000000),vel1,z0,Extruder\WObj:=Workobject_1;
MoveL RelTool (p1,67.356880,16.000000,6.758109,\Rx:=0.000000,\Ry:=0.000000),vel1,z0,Extruder\WObj:=Workobject_1;
MoveL RelTool (p1,66.615646,16.000000,7.074461,\Rx:=0.000000,\Ry:=0.000000),vel1,z0,Extruder\WObj:=Workobject_1;
MoveL RelTool (p1,65.934883,16.000000,7.505786,\Rx:=0.000000,\Ry:=0.000000),vel1,z0,Extruder\WObj:=Workobject_1;
MoveL RelTool (p1,65.332253,16.000000,8.040880,\Rx:=0.000000,\Ry:=0.000000),vel1,z0,Extruder\WObj:=Workobject_1;
MoveL RelTool (p1,64.823410,16.000000,8.665841,\Rx:=0.000000,\Ry:=0.000000),vel1,z0,Extruder\WObj:=Workobject_1;
MoveL RelTool (p1,64.363686,16.000000,9.273595,\Rx:=0.000000,\Ry:=0.000000),vel1,z0,Extruder\WObj:=Workobject_1;
MoveL RelTool (p1,63.963219,16.000000,9.720532,\Rx:=0.000000,\Ry:=0.000000),vel1,z0,Extruder\WObj:=Workobject_1;
MoveL RelTool (p1,63.821823,16.000000,9.878342,\Rx:=0.000000,\Ry:=0.000000),vel1,z0,Extruder\WObj:=Workobject_1;
MoveL RelTool (p1,63.165062,16.000000,10.507496,\Rx:=0.000000,\Ry:=0.000000),vel1,z0,Extruder\WObj:=Workobject_1;
MoveL RelTool (p1,62.831947,16.000000,10.783607,\Rx:=0.000000,\Ry:=0.000000),vel1,z0,Extruder\WObj:=Workobject_1;
MoveL RelTool (p1,62.416321,16.000000,11.128095,\Rx:=0.000000,\Ry:=0.000000),vel1,z0,Extruder\WObj:=Workobject_1;
MoveL RelTool (p1,61.578415,16.000000,11.733726,\Rx:=0.000000,\Ry:=0.000000),vel1,z0,Extruder\WObj:=Workobject_1;
MoveL RelTool (p1,61.418831,16.000000,11.834675,\Rx:=0.000000,\Ry:=0.000000),vel1,z0,Extruder\WObj:=Workobject_1;
MoveL RelTool (p1,60.616638,16.000000,12.342117,\Rx:=0.000000,\Ry:=0.000000),vel1,z0,Extruder\WObj:=Workobject_1;
MoveL RelTool (p1,59.722591,16.000000,12.837377,\Rx:=0.000000,\Ry:=0.000000),vel1,z0,Extruder\WObj:=Workobject_1;
MoveL RelTool (p1,59.593624,16.000000,12.908818,\Rx:=0.000000,\Ry:=0.000000),vel1,z0,Extruder\WObj:=Workobject_1;
MoveL RelTool (p1,58.474972,16.000000,13.452054,\Rx:=0.000000,\Ry:=0.000000),vel1,z0,Extruder\WObj:=Workobject_1;
MoveL RelTool (p1,57.753036,16.000000,13.758680,\Rx:=0.000000,\Ry:=0.000000),vel1,z0,Extruder\WObj:=Workobject_1;
MoveL RelTool (p1,57.254681,16.000000,13.970348,\Rx:=0.000000,\Ry:=0.000000),vel1,z0,Extruder\WObj:=Workobject_1;
MoveL RelTool (p1,55.907604,16.000000,14.468318,\Rx:=0.000000,\Ry:=0.000000),vel1,z0,Extruder\WObj:=Workobject_1;
MoveL RelTool (p1,55.501736,16.000000,14.597532,\Rx:=0.000000,\Ry:=0.000000),vel1,z0,Extruder\WObj:=Workobject_1;
MoveL RelTool (p1,54.486706,16.000000,14.920681,\Rx:=0.000000,\Ry:=0.000000),vel1,z0,Extruder\WObj:=Workobject_1;
MoveL RelTool (p1,53.019268,16.000000,15.316940,\Rx:=0.000000,\Ry:=0.000000),vel1,z0,Extruder\WObj:=Workobject_1;
MoveL RelTool (p1,52.986862,16.000000,15.324217,\Rx:=0.000000,\Ry:=0.000000),vel1,z0,Extruder\WObj:=Workobject_1;
MoveL RelTool (p1,51.488445,16.000000,15.660700,\Rx:=0.000000,\Ry:=0.000000),vel1,z0,Extruder\WObj:=Workobject_1;
MoveL RelTool (p1,50.290966,16.000000,15.877948,\Rx:=0.000000,\Ry:=0.000000),vel1,z0,Extruder\WObj:=Workobject_1;
MoveL RelTool (p1,49.889133,16.000000,15.950849,\Rx:=0.000000,\Ry:=0.000000),vel1,z0,Extruder\WObj:=Workobject_1;
MoveL RelTool (p1,48.224419,16.000000,16.184232,\Rx:=0.000000,\Ry:=0.000000),vel1,z0,Extruder\WObj:=Workobject_1;
MoveL RelTool (p1,47.446861,16.000000,16.262141,\Rx:=0.000000,\Ry:=0.000000),vel1,z0,Extruder\WObj:=Workobject_1;
MoveL RelTool (p1,46.521641,16.000000,16.354847,\Rx:=0.000000,\Ry:=0.000000),vel1,z0,Extruder\WObj:=Workobject_1;
MoveL RelTool (p1,44.783478,16.000000,16.461150,\Rx:=0.000000,\Ry:=0.000000),vel1,z0,Extruder\WObj:=Workobject_1;
MoveL RelTool (p1,44.466858,16.000000,16.468186,\Rx:=0.000000,\Ry:=0.000000),vel1,z0,Extruder\WObj:=Workobject_1;
MoveL RelTool (p1,43.043808,16.000000,16.499818,\Rx:=0.000000,\Ry:=0.000000),vel1,z0,Extruder\WObj:=Workobject_1;
MoveL RelTool (p1,41.456497,16.000000,16.473560,\Rx:=0.000000,\Ry:=0.000000),vel1,z0,Extruder\WObj:=Workobject_1;
MoveL RelTool (p1,41.303349,16.000000,16.471027,\Rx:=0.000000,\Ry:=0.000000),vel1,z0,Extruder\WObj:=Workobject_1;
MoveL RelTool (p1,39.566307,16.000000,16.374732,\Rx:=0.000000,\Ry:=0.000000),vel1,z0,Extruder\WObj:=Workobject_1;
MoveL RelTool (p1,38.468281,16.000000,16.271000,\Rx:=0.000000,\Ry:=0.000000),vel1,z0,Extruder\WObj:=Workobject_1;
MoveL RelTool (p1,37.849564,16.000000,16.212550,\Rx:=0.000000,\Ry:=0.000000),vel1,z0,Extruder\WObj:=Workobject_1;
MoveL RelTool (p1,36.162739,16.000000,15.985516,\Rx:=0.000000,\Ry:=0.000000),vel1,z0,Extruder\WObj:=Workobject_1;
MoveL RelTool (p1,35.548347,16.000000,15.877330,\Rx:=0.000000,\Ry:=0.000000),vel1,z0,Extruder\WObj:=Workobject_1;
MoveL RelTool (p1,34.531830,16.000000,15.698334,\Rx:=0.000000,\Ry:=0.000000),vel1,z0,Extruder\WObj:=Workobject_1;
MoveL RelTool (p1,32.962124,16.000000,15.353427,\Rx:=0.000000,\Ry:=0.000000),vel1,z0,Extruder\WObj:=Workobject_1;
MoveL RelTool (p1,32.770821,16.000000,15.302555,\Rx:=0.000000,\Ry:=0.000000),vel1,z0,Extruder\WObj:=Workobject_1;
MoveL RelTool (p1,31.457693,16.000000,14.953369,\Rx:=0.000000,\Ry:=0.000000),vel1,z0,Extruder\WObj:=Workobject_1;
MoveL RelTool (p1,30.226080,16.000000,14.565704,\Rx:=0.000000,\Ry:=0.000000),vel1,z0,Extruder\WObj:=Workobject_1;
MoveL RelTool (p1,30.018776,16.000000,14.500453,\Rx:=0.000000,\Ry:=0.000000),vel1,z0,Extruder\WObj:=Workobject_1;
MoveL RelTool (p1,28.659712,16.000000,14.002768,\Rx:=0.000000,\Ry:=0.000000),vel1,z0,Extruder\WObj:=Workobject_1;
MoveL RelTool (p1,27.918875,16.000000,13.690347,\Rx:=0.000000,\Ry:=0.000000),vel1,z0,Extruder\WObj:=Workobject_1;
MoveL RelTool (p1,27.404802,16.000000,13.473557,\Rx:=0.000000,\Ry:=0.000000),vel1,z0,Extruder\WObj:=Workobject_1;
MoveL RelTool (p1,26.235151,16.000000,12.906940,\Rx:=0.000000,\Ry:=0.000000),vel1,z0,Extruder\WObj:=Workobject_1;
MoveL RelTool (p1,25.867798,16.000000,12.702785,\Rx:=0.000000,\Ry:=0.000000),vel1,z0,Extruder\WObj:=Workobject_1;
MoveL RelTool (p1,25.171089,16.000000,12.315596,\Rx:=0.000000,\Ry:=0.000000),vel1,z0,Extruder\WObj:=Workobject_1;
MoveL RelTool (p1,24.206091,16.000000,11.701200,\Rx:=0.000000,\Ry:=0.000000),vel1,z0,Extruder\WObj:=Workobject_1;
MoveL RelTool (p1,24.143076,16.000000,11.655322,\Rx:=0.000000,\Ry:=0.000000),vel1,z0,Extruder\WObj:=Workobject_1;
MoveL RelTool (p1,23.372747,16.000000,11.094489,\Rx:=0.000000,\Ry:=0.000000),vel1,z0,Extruder\WObj:=Workobject_1;
MoveL RelTool (p1,22.748590,16.000000,10.572390,\Rx:=0.000000,\Ry:=0.000000),vel1,z0,Extruder\WObj:=Workobject_1;
MoveL RelTool (p1,22.615110,16.000000,10.460735,\Rx:=0.000000,\Ry:=0.000000),vel1,z0,Extruder\WObj:=Workobject_1;
MoveL RelTool (p1,21.967155,16.000000,9.833263,\Rx:=0.000000,\Ry:=0.000000),vel1,z0,Extruder\WObj:=Workobject_1;
MoveL RelTool (p1,21.661156,16.000000,9.486848,\Rx:=0.000000,\Ry:=0.000000),vel1,z0,Extruder\WObj:=Workobject_1;
MoveL RelTool (p1,21.416798,16.000000,9.210219,\Rx:=0.000000,\Ry:=0.000000),vel1,z0,Extruder\WObj:=Workobject_1;
MoveL RelTool (p1,21.008959,16.000000,8.665841,\Rx:=0.000000,\Ry:=0.000000),vel1,z0,Extruder\WObj:=Workobject_1;
MoveL RelTool (p1,20.500122,16.000000,8.040880,\Rx:=0.000000,\Ry:=0.000000),vel1,z0,Extruder\WObj:=Workobject_1;
MoveL RelTool (p1,19.897491,16.000000,7.505786,\Rx:=0.000000,\Ry:=0.000000),vel1,z0,Extruder\WObj:=Workobject_1;
MoveL RelTool (p1,19.216721,16.000000,7.074461,\Rx:=0.000000,\Ry:=0.000000),vel1,z0,Extruder\WObj:=Workobject_1;
MoveL RelTool (p1,18.475496,16.000000,6.758109,\Rx:=0.000000,\Ry:=0.000000),vel1,z0,Extruder\WObj:=Workobject_1;
MoveL RelTool (p1,17.693081,16.000000,6.564949,\Rx:=0.000000,\Ry:=0.000000),vel1,z0,Extruder\WObj:=Workobject_1;
MoveL RelTool (p1,16.889791,16.000000,6.500000,\Rx:=0.000000,\Ry:=0.000000),vel1,z0,Extruder\WObj:=Workobject_1;
MoveL RelTool (p1,3.000000,16.000000,6.500000,\Rx:=0.000000,\Ry:=0.000000),vel1,z0,Extruder\WObj:=Workobject_1;
MoveL RelTool (p1,3.000000,3.000000,6.500000,\Rx:=0.000000,\Ry:=0.000000),vel1,z0,Extruder\WObj:=Workobject_1;


MoveL RelTool (p1,3.000000,3.000000,6.500000,\Rx:=0.000000,\Ry:=0),vel1,zoneval,Extruder\WObj:=Workobject_1;
MoveL RelTool (p1,5.000000,3.000000,6.500000,\Rx:=0.000000,\Ry:=-0.000000),vel1,zoneval,Extruder\WObj:=Workobject_1;
MoveL RelTool (p1,7.500000,3.000000,6.500000,\Rx:=0.000000,\Ry:=-0.000000),vel1,zoneval,Extruder\WObj:=Workobject_1;
MoveL RelTool (p1,10.000000,3.000000,6.500000,\Rx:=0.000000,\Ry:=-0.000000),vel1,zoneval,Extruder\WObj:=Workobject_1;
MoveL RelTool (p1,12.500000,3.000000,6.500000,\Rx:=0.000000,\Ry:=-0.000000),vel1,zoneval,Extruder\WObj:=Workobject_1;
MoveL RelTool (p1,15.000000,3.000000,6.500000,\Rx:=0.000000,\Ry:=-0.000000),vel1,zoneval,Extruder\WObj:=Workobject_1;
MoveL RelTool (p1,17.500000,3.000000,6.549338,\Rx:=0.000000,\Ry:=-2.301628),vel1,zoneval,Extruder\WObj:=Workobject_1;
MoveL RelTool (p1,20.000000,3.000000,7.596807,\Rx:=0.000000,\Ry:=-9.245074),vel1,zoneval,Extruder\WObj:=Workobject_1;
MoveL RelTool (p1,22.500000,3.000000,10.332328,\Rx:=0.000000,\Ry:=-9.203115),vel1,zoneval,Extruder\WObj:=Workobject_1;
MoveL RelTool (p1,25.000000,3.000000,12.181567,\Rx:=0.000000,\Ry:=-6.983793),vel1,zoneval,Extruder\WObj:=Workobject_1;
MoveL RelTool (p1,27.500000,3.000000,13.497451,\Rx:=0.000000,\Ry:=-5.532306),vel1,zoneval,Extruder\WObj:=Workobject_1;
MoveL RelTool (p1,30.000000,3.000000,14.484560,\Rx:=0.000000,\Ry:=-4.046642),vel1,zoneval,Extruder\WObj:=Workobject_1;
MoveL RelTool (p1,32.500000,3.000000,15.227603,\Rx:=0.000000,\Ry:=-3.145456),vel1,zoneval,Extruder\WObj:=Workobject_1;
MoveL RelTool (p1,35.000000,3.000000,15.771037,\Rx:=0.000000,\Ry:=-2.619262),vel1,zoneval,Extruder\WObj:=Workobject_1;
MoveL RelTool (p1,37.500000,3.000000,16.148328,\Rx:=0.000000,\Ry:=-1.705318),vel1,zoneval,Extruder\WObj:=Workobject_1;
MoveL RelTool (p1,40.000000,3.000000,16.379958,\Rx:=0.000000,\Ry:=-0.840101),vel1,zoneval,Extruder\WObj:=Workobject_1;
MoveL RelTool (p1,42.500000,3.000000,16.475136,\Rx:=0.000000,\Ry:=0.012935),vel1,zoneval,Extruder\WObj:=Workobject_1;
MoveL RelTool (p1,45.000000,3.000000,16.436871,\Rx:=0.000000,\Ry:=0.864966),vel1,zoneval,Extruder\WObj:=Workobject_1;
MoveL RelTool (p1,47.500000,3.000000,16.263228,\Rx:=0.000000,\Ry:=1.718686),vel1,zoneval,Extruder\WObj:=Workobject_1;
MoveL RelTool (p1,50.000000,3.000000,15.923700,\Rx:=0.000000,\Ry:=2.090726),vel1,zoneval,Extruder\WObj:=Workobject_1;
MoveL RelTool (p1,52.500000,3.000000,15.425496,\Rx:=0.000000,\Ry:=2.632317),vel1,zoneval,Extruder\WObj:=Workobject_1;
MoveL RelTool (p1,55.000000,3.000000,14.747982,\Rx:=0.000000,\Ry:=3.550580),vel1,zoneval,Extruder\WObj:=Workobject_1;
MoveL RelTool (p1,57.500000,3.000000,13.860923,\Rx:=0.000000,\Ry:=5.062336),vel1,zoneval,Extruder\WObj:=Workobject_1;
MoveL RelTool (p1,60.000000,3.000000,12.677522,\Rx:=0.000000,\Ry:=6.787941),vel1,zoneval,Extruder\WObj:=Workobject_1;
MoveL RelTool (p1,62.500000,3.000000,11.039633,\Rx:=0.000000,\Ry:=8.641351),vel1,zoneval,Extruder\WObj:=Workobject_1;
MoveL RelTool (p1,65.000000,3.000000,8.448953,\Rx:=0.000000,\Ry:=10.686183),vel1,zoneval,Extruder\WObj:=Workobject_1;
MoveL RelTool (p1,67.500000,3.000000,6.722776,\Rx:=0.000000,\Ry:=3.081723),vel1,zoneval,Extruder\WObj:=Workobject_1;
MoveL RelTool (p1,70.000000,3.000000,6.500000,\Rx:=0.000000,\Ry:=-0.000000),vel1,zoneval,Extruder\WObj:=Workobject_1;
MoveL RelTool (p1,72.500000,3.000000,6.500000,\Rx:=0.000000,\Ry:=-0.000000),vel1,zoneval,Extruder\WObj:=Workobject_1;
MoveL RelTool (p1,75.000000,3.000000,6.500000,\Rx:=0.000000,\Ry:=-0.000000),vel1,zoneval,Extruder\WObj:=Workobject_1;
MoveL RelTool (p1,77.500000,3.000000,6.500000,\Rx:=0.000000,\Ry:=-0.000000),vel1,zoneval,Extruder\WObj:=Workobject_1;
MoveL RelTool (p1,80.000000,3.000000,6.500000,\Rx:=0.000000,\Ry:=-0.000000),vel1,zoneval,Extruder\WObj:=Workobject_1;
MoveL RelTool (p1,82.500000,3.000000,6.500000,\Rx:=0.000000,\Ry:=-0.000000),vel1,zoneval,Extruder\WObj:=Workobject_1;
MoveL RelTool (p1,80.500000,3.500000,6.500000,\Rx:=0.000000,\Ry:=0.000000),vel1,zoneval,Extruder\WObj:=Workobject_1;
MoveL RelTool (p1,78.000000,3.500000,6.500000,\Rx:=0.000000,\Ry:=0.000000),vel1,zoneval,Extruder\WObj:=Workobject_1;
MoveL RelTool (p1,75.500000,3.500000,6.500000,\Rx:=0.000000,\Ry:=0.000000),vel1,zoneval,Extruder\WObj:=Workobject_1;
MoveL RelTool (p1,73.000000,3.500000,6.500000,\Rx:=0.000000,\Ry:=0.000000),vel1,zoneval,Extruder\WObj:=Workobject_1;
MoveL RelTool (p1,70.500000,3.500000,6.500000,\Rx:=0.000000,\Ry:=0.000000),vel1,zoneval,Extruder\WObj:=Workobject_1;
MoveL RelTool (p1,68.000000,3.500000,6.599337,\Rx:=0.000000,\Ry:=3.081723),vel1,zoneval,Extruder\WObj:=Workobject_1;
MoveL RelTool (p1,65.500000,3.500000,7.891932,\Rx:=0.000000,\Ry:=10.686183),vel1,zoneval,Extruder\WObj:=Workobject_1;
MoveL RelTool (p1,63.000000,3.500000,10.637015,\Rx:=0.000000,\Ry:=8.638332),vel1,zoneval,Extruder\WObj:=Workobject_1;
MoveL RelTool (p1,60.500000,3.500000,12.383557,\Rx:=0.000000,\Ry:=6.787941),vel1,zoneval,Extruder\WObj:=Workobject_1;
MoveL RelTool (p1,58.000000,3.500000,13.651217,\Rx:=0.000000,\Ry:=5.071485),vel1,zoneval,Extruder\WObj:=Workobject_1;
MoveL RelTool (p1,55.500000,3.500000,14.604676,\Rx:=0.000000,\Ry:=3.553825),vel1,zoneval,Extruder\WObj:=Workobject_1;
MoveL RelTool (p1,53.000000,3.500000,15.320621,\Rx:=0.000000,\Ry:=2.656042),vel1,zoneval,Extruder\WObj:=Workobject_1;
MoveL RelTool (p1,50.500000,3.500000,15.841818,\Rx:=0.000000,\Ry:=2.078299),vel1,zoneval,Extruder\WObj:=Workobject_1;
MoveL RelTool (p1,48.000000,3.500000,16.195787,\Rx:=0.000000,\Ry:=1.723243),vel1,zoneval,Extruder\WObj:=Workobject_1;
MoveL RelTool (p1,45.500000,3.500000,16.403679,\Rx:=0.000000,\Ry:=0.864966),vel1,zoneval,Extruder\WObj:=Workobject_1;
MoveL RelTool (p1,43.000000,3.500000,16.475599,\Rx:=0.000000,\Ry:=0.012935),vel1,zoneval,Extruder\WObj:=Workobject_1;
MoveL RelTool (p1,40.500000,3.500000,16.413898,\Rx:=0.000000,\Ry:=-0.840101),vel1,zoneval,Extruder\WObj:=Workobject_1;
MoveL RelTool (p1,38.000000,3.500000,16.216357,\Rx:=0.000000,\Ry:=-1.705318),vel1,zoneval,Extruder\WObj:=Workobject_1;
MoveL RelTool (p1,35.500000,3.500000,15.876245,\Rx:=0.000000,\Ry:=-2.633413),vel1,zoneval,Extruder\WObj:=Workobject_1;
MoveL RelTool (p1,33.000000,3.500000,15.353994,\Rx:=0.000000,\Ry:=-3.127352),vel1,zoneval,Extruder\WObj:=Workobject_1;
MoveL RelTool (p1,30.500000,3.500000,14.650097,\Rx:=0.000000,\Ry:=-4.062966),vel1,zoneval,Extruder\WObj:=Workobject_1;
MoveL RelTool (p1,28.000000,3.500000,13.729833,\Rx:=0.000000,\Ry:=-5.524357),vel1,zoneval,Extruder\WObj:=Workobject_1;
MoveL RelTool (p1,25.500000,3.500000,12.488227,\Rx:=0.000000,\Ry:=-6.983793),vel1,zoneval,Extruder\WObj:=Workobject_1;
MoveL RelTool (p1,23.000000,3.500000,10.774609,\Rx:=0.000000,\Ry:=-9.213373),vel1,zoneval,Extruder\WObj:=Workobject_1;
MoveL RelTool (p1,20.500000,3.500000,8.040772,\Rx:=0.000000,\Ry:=-9.245074),vel1,zoneval,Extruder\WObj:=Workobject_1;
MoveL RelTool (p1,18.000000,3.500000,6.640720,\Rx:=0.000000,\Ry:=-2.301628),vel1,zoneval,Extruder\WObj:=Workobject_1;
MoveL RelTool (p1,15.500000,3.500000,6.500000,\Rx:=0.000000,\Ry:=0.000000),vel1,zoneval,Extruder\WObj:=Workobject_1;
MoveL RelTool (p1,13.000000,3.500000,6.500000,\Rx:=0.000000,\Ry:=0.000000),vel1,zoneval,Extruder\WObj:=Workobject_1;
MoveL RelTool (p1,10.500000,3.500000,6.500000,\Rx:=0.000000,\Ry:=0.000000),vel1,zoneval,Extruder\WObj:=Workobject_1;
MoveL RelTool (p1,8.000000,3.500000,6.500000,\Rx:=0.000000,\Ry:=0.000000),vel1,zoneval,Extruder\WObj:=Workobject_1;
MoveL RelTool (p1,5.500000,3.500000,6.500000,\Rx:=0.000000,\Ry:=0.000000),vel1,zoneval,Extruder\WObj:=Workobject_1;
MoveL RelTool (p1,3.000000,3.500000,6.500000,\Rx:=0.000000,\Ry:=0.000000),vel1,zoneval,Extruder\WObj:=Workobject_1;
MoveL RelTool (p1,5.000000,4.000000,6.500000,\Rx:=0.000000,\Ry:=-0.000000),vel1,zoneval,Extruder\WObj:=Workobject_1;
MoveL RelTool (p1,7.500000,4.000000,6.500000,\Rx:=0.000000,\Ry:=-0.000000),vel1,zoneval,Extruder\WObj:=Workobject_1;
MoveL RelTool (p1,10.000000,4.000000,6.500000,\Rx:=0.000000,\Ry:=-0.000000),vel1,zoneval,Extruder\WObj:=Workobject_1;
MoveL RelTool (p1,12.500000,4.000000,6.500000,\Rx:=0.000000,\Ry:=-0.000000),vel1,zoneval,Extruder\WObj:=Workobject_1;
MoveL RelTool (p1,15.000000,4.000000,6.500000,\Rx:=0.000000,\Ry:=-0.000000),vel1,zoneval,Extruder\WObj:=Workobject_1;
MoveL RelTool (p1,17.500000,4.000000,6.549338,\Rx:=0.000000,\Ry:=-2.301628),vel1,zoneval,Extruder\WObj:=Workobject_1;
MoveL RelTool (p1,20.000000,4.000000,7.596807,\Rx:=0.000000,\Ry:=-9.245074),vel1,zoneval,Extruder\WObj:=Workobject_1;
MoveL RelTool (p1,22.500000,4.000000,10.333402,\Rx:=0.000000,\Ry:=-9.223617),vel1,zoneval,Extruder\WObj:=Workobject_1;
MoveL RelTool (p1,25.000000,4.000000,12.183835,\Rx:=0.000000,\Ry:=-6.983793),vel1,zoneval,Extruder\WObj:=Workobject_1;
MoveL RelTool (p1,27.500000,4.000000,13.498887,\Rx:=0.000000,\Ry:=-5.534830),vel1,zoneval,Extruder\WObj:=Workobject_1;
MoveL RelTool (p1,30.000000,4.000000,14.485238,\Rx:=0.000000,\Ry:=-4.079275),vel1,zoneval,Extruder\WObj:=Workobject_1;
MoveL RelTool (p1,32.500000,4.000000,15.229702,\Rx:=0.000000,\Ry:=-3.109236),vel1,zoneval,Extruder\WObj:=Workobject_1;
MoveL RelTool (p1,35.000000,4.000000,15.771624,\Rx:=0.000000,\Ry:=-2.627103),vel1,zoneval,Extruder\WObj:=Workobject_1;
MoveL RelTool (p1,37.500000,4.000000,16.149645,\Rx:=0.000000,\Ry:=-1.705318),vel1,zoneval,Extruder\WObj:=Workobject_1;
MoveL RelTool (p1,40.000000,4.000000,16.381760,\Rx:=0.000000,\Ry:=-0.840101),vel1,zoneval,Extruder\WObj:=Workobject_1;
MoveL RelTool (p1,42.500000,4.000000,16.477077,\Rx:=0.000000,\Ry:=0.012935),vel1,zoneval,Extruder\WObj:=Workobject_1;
MoveL RelTool (p1,45.000000,4.000000,16.438525,\Rx:=0.000000,\Ry:=0.864966),vel1,zoneval,Extruder\WObj:=Workobject_1;
MoveL RelTool (p1,47.500000,4.000000,16.264455,\Rx:=0.000000,\Ry:=1.726103),vel1,zoneval,Extruder\WObj:=Workobject_1;
MoveL RelTool (p1,50.000000,4.000000,15.924630,\Rx:=0.000000,\Ry:=2.065868),vel1,zoneval,Extruder\WObj:=Workobject_1;
MoveL RelTool (p1,52.500000,4.000000,15.427429,\Rx:=0.000000,\Ry:=2.679747),vel1,zoneval,Extruder\WObj:=Workobject_1;
MoveL RelTool (p1,55.000000,4.000000,14.747969,\Rx:=0.000000,\Ry:=3.559873),vel1,zoneval,Extruder\WObj:=Workobject_1;
MoveL RelTool (p1,57.500000,4.000000,13.862318,\Rx:=0.000000,\Ry:=5.080628),vel1,zoneval,Extruder\WObj:=Workobject_1;
MoveL RelTool (p1,60.000000,4.000000,12.679713,\Rx:=0.000000,\Ry:=6.787941),vel1,zoneval,Extruder\WObj:=Workobject_1;
MoveL RelTool (p1,62.500000,4.000000,11.040504,\Rx:=0.000000,\Ry:=8.635312),vel1,zoneval,Extruder\WObj:=Workobject_1;
MoveL RelTool (p1,65.000000,4.000000,8.448953,\Rx:=0.000000,\Ry:=10.686183),vel1,zoneval,Extruder\WObj:=Workobject_1;
MoveL RelTool (p1,67.500000,4.000000,6.722776,\Rx:=0.000000,\Ry:=3.081723),vel1,zoneval,Extruder\WObj:=Workobject_1;
MoveL RelTool (p1,70.000000,4.000000,6.500000,\Rx:=0.000000,\Ry:=-0.000000),vel1,zoneval,Extruder\WObj:=Workobject_1;
MoveL RelTool (p1,72.500000,4.000000,6.500000,\Rx:=0.000000,\Ry:=-0.000000),vel1,zoneval,Extruder\WObj:=Workobject_1;
MoveL RelTool (p1,75.000000,4.000000,6.500000,\Rx:=0.000000,\Ry:=-0.000000),vel1,zoneval,Extruder\WObj:=Workobject_1;
MoveL RelTool (p1,77.500000,4.000000,6.500000,\Rx:=0.000000,\Ry:=-0.000000),vel1,zoneval,Extruder\WObj:=Workobject_1;
MoveL RelTool (p1,80.000000,4.000000,6.500000,\Rx:=0.000000,\Ry:=-0.000000),vel1,zoneval,Extruder\WObj:=Workobject_1;
MoveL RelTool (p1,82.500000,4.000000,6.500000,\Rx:=0.000000,\Ry:=-0.000000),vel1,zoneval,Extruder\WObj:=Workobject_1;
MoveL RelTool (p1,80.500000,4.500000,6.500000,\Rx:=0.000000,\Ry:=0.000000),vel1,zoneval,Extruder\WObj:=Workobject_1;
MoveL RelTool (p1,78.000000,4.500000,6.500000,\Rx:=0.000000,\Ry:=0.000000),vel1,zoneval,Extruder\WObj:=Workobject_1;
MoveL RelTool (p1,75.500000,4.500000,6.500000,\Rx:=0.000000,\Ry:=0.000000),vel1,zoneval,Extruder\WObj:=Workobject_1;
MoveL RelTool (p1,73.000000,4.500000,6.500000,\Rx:=0.000000,\Ry:=0.000000),vel1,zoneval,Extruder\WObj:=Workobject_1;
MoveL RelTool (p1,70.500000,4.500000,6.500000,\Rx:=0.000000,\Ry:=0.000000),vel1,zoneval,Extruder\WObj:=Workobject_1;
MoveL RelTool (p1,68.000000,4.500000,6.599337,\Rx:=0.000000,\Ry:=3.081723),vel1,zoneval,Extruder\WObj:=Workobject_1;
MoveL RelTool (p1,65.500000,4.500000,7.891932,\Rx:=0.000000,\Ry:=10.686183),vel1,zoneval,Extruder\WObj:=Workobject_1;
MoveL RelTool (p1,63.000000,4.500000,10.638278,\Rx:=0.000000,\Ry:=8.632290),vel1,zoneval,Extruder\WObj:=Workobject_1;
MoveL RelTool (p1,60.500000,4.500000,12.385749,\Rx:=0.000000,\Ry:=6.787941),vel1,zoneval,Extruder\WObj:=Workobject_1;
MoveL RelTool (p1,58.000000,4.500000,13.651767,\Rx:=0.000000,\Ry:=5.089766),vel1,zoneval,Extruder\WObj:=Workobject_1;
MoveL RelTool (p1,55.500000,4.500000,14.604149,\Rx:=0.000000,\Ry:=3.565919),vel1,zoneval,Extruder\WObj:=Workobject_1;
MoveL RelTool (p1,53.000000,4.500000,15.320607,\Rx:=0.000000,\Ry:=2.703434),vel1,zoneval,Extruder\WObj:=Workobject_1;
MoveL RelTool (p1,50.500000,4.500000,15.843750,\Rx:=0.000000,\Ry:=2.053433),vel1,zoneval,Extruder\WObj:=Workobject_1;
MoveL RelTool (p1,48.000000,4.500000,16.196717,\Rx:=0.000000,\Ry:=1.706516),vel1,zoneval,Extruder\WObj:=Workobject_1;
MoveL RelTool (p1,45.500000,4.500000,16.405333,\Rx:=0.000000,\Ry:=0.864966),vel1,zoneval,Extruder\WObj:=Workobject_1;
MoveL RelTool (p1,43.000000,4.500000,16.477540,\Rx:=0.000000,\Ry:=0.012935),vel1,zoneval,Extruder\WObj:=Workobject_1;
MoveL RelTool (p1,40.500000,4.500000,16.415700,\Rx:=0.000000,\Ry:=-0.840101),vel1,zoneval,Extruder\WObj:=Workobject_1;
MoveL RelTool (p1,38.000000,4.500000,16.217674,\Rx:=0.000000,\Ry:=-1.705318),vel1,zoneval,Extruder\WObj:=Workobject_1;
MoveL RelTool (p1,35.500000,4.500000,15.875969,\Rx:=0.000000,\Ry:=-2.612354),vel1,zoneval,Extruder\WObj:=Workobject_1;
MoveL RelTool (p1,33.000000,4.500000,15.354581,\Rx:=0.000000,\Ry:=-3.091107),vel1,zoneval,Extruder\WObj:=Workobject_1;
MoveL RelTool (p1,30.500000,4.500000,14.652196,\Rx:=0.000000,\Ry:=-4.095571),vel1,zoneval,Extruder\WObj:=Workobject_1;
MoveL RelTool (p1,28.000000,4.500000,13.732216,\Rx:=0.000000,\Ry:=-5.544211),vel1,zoneval,Extruder\WObj:=Workobject_1;
MoveL RelTool (p1,25.500000,4.500000,12.490495,\Rx:=0.000000,\Ry:=-6.983793),vel1,zoneval,Extruder\WObj:=Workobject_1;
MoveL RelTool (p1,23.000000,4.500000,10.777117,\Rx:=0.000000,\Ry:=-9.233845),vel1,zoneval,Extruder\WObj:=Workobject_1;
MoveL RelTool (p1,20.500000,4.500000,8.040772,\Rx:=0.000000,\Ry:=-9.245074),vel1,zoneval,Extruder\WObj:=Workobject_1;
MoveL RelTool (p1,18.000000,4.500000,6.640720,\Rx:=0.000000,\Ry:=-2.301628),vel1,zoneval,Extruder\WObj:=Workobject_1;
MoveL RelTool (p1,15.500000,4.500000,6.500000,\Rx:=0.000000,\Ry:=0.000000),vel1,zoneval,Extruder\WObj:=Workobject_1;
MoveL RelTool (p1,13.000000,4.500000,6.500000,\Rx:=0.000000,\Ry:=0.000000),vel1,zoneval,Extruder\WObj:=Workobject_1;
MoveL RelTool (p1,10.500000,4.500000,6.500000,\Rx:=0.000000,\Ry:=0.000000),vel1,zoneval,Extruder\WObj:=Workobject_1;
MoveL RelTool (p1,8.000000,4.500000,6.500000,\Rx:=0.000000,\Ry:=0.000000),vel1,zoneval,Extruder\WObj:=Workobject_1;
MoveL RelTool (p1,5.500000,4.500000,6.500000,\Rx:=0.000000,\Ry:=0.000000),vel1,zoneval,Extruder\WObj:=Workobject_1;
MoveL RelTool (p1,3.000000,4.500000,6.500000,\Rx:=0.000000,\Ry:=0.000000),vel1,zoneval,Extruder\WObj:=Workobject_1;
MoveL RelTool (p1,5.000000,5.000000,6.500000,\Rx:=0.000000,\Ry:=-0.000000),vel1,zoneval,Extruder\WObj:=Workobject_1;
MoveL RelTool (p1,7.500000,5.000000,6.500000,\Rx:=0.000000,\Ry:=-0.000000),vel1,zoneval,Extruder\WObj:=Workobject_1;
MoveL RelTool (p1,10.000000,5.000000,6.500000,\Rx:=0.000000,\Ry:=-0.000000),vel1,zoneval,Extruder\WObj:=Workobject_1;
MoveL RelTool (p1,12.500000,5.000000,6.500000,\Rx:=0.000000,\Ry:=-0.000000),vel1,zoneval,Extruder\WObj:=Workobject_1;
MoveL RelTool (p1,15.000000,5.000000,6.500000,\Rx:=0.000000,\Ry:=-0.000000),vel1,zoneval,Extruder\WObj:=Workobject_1;
MoveL RelTool (p1,17.500000,5.000000,6.549338,\Rx:=0.000000,\Ry:=-2.301628),vel1,zoneval,Extruder\WObj:=Workobject_1;
MoveL RelTool (p1,20.000000,5.000000,7.596807,\Rx:=0.000000,\Ry:=-9.245074),vel1,zoneval,Extruder\WObj:=Workobject_1;
MoveL RelTool (p1,22.500000,5.000000,10.334477,\Rx:=0.000000,\Ry:=-9.244059),vel1,zoneval,Extruder\WObj:=Workobject_1;
MoveL RelTool (p1,25.000000,5.000000,12.186103,\Rx:=0.000000,\Ry:=-6.983793),vel1,zoneval,Extruder\WObj:=Workobject_1;
MoveL RelTool (p1,27.500000,5.000000,13.500323,\Rx:=0.000000,\Ry:=-5.522195),vel1,zoneval,Extruder\WObj:=Workobject_1;
MoveL RelTool (p1,30.000000,5.000000,14.485915,\Rx:=0.000000,\Ry:=-4.111853),vel1,zoneval,Extruder\WObj:=Workobject_1;
MoveL RelTool (p1,32.500000,5.000000,15.231801,\Rx:=0.000000,\Ry:=-3.072965),vel1,zoneval,Extruder\WObj:=Workobject_1;
MoveL RelTool (p1,35.000000,5.000000,15.772211,\Rx:=0.000000,\Ry:=-2.597598),vel1,zoneval,Extruder\WObj:=Workobject_1;
MoveL RelTool (p1,37.500000,5.000000,16.150962,\Rx:=0.000000,\Ry:=-1.705318),vel1,zoneval,Extruder\WObj:=Workobject_1;
MoveL RelTool (p1,40.000000,5.000000,16.383563,\Rx:=0.000000,\Ry:=-0.840101),vel1,zoneval,Extruder\WObj:=Workobject_1;
MoveL RelTool (p1,42.500000,5.000000,16.479018,\Rx:=0.000000,\Ry:=0.012935),vel1,zoneval,Extruder\WObj:=Workobject_1;
MoveL RelTool (p1,45.000000,5.000000,16.440180,\Rx:=0.000000,\Ry:=0.864966),vel1,zoneval,Extruder\WObj:=Workobject_1;
MoveL RelTool (p1,47.500000,5.000000,16.263818,\Rx:=0.000000,\Ry:=1.686921),vel1,zoneval,Extruder\WObj:=Workobject_1;
MoveL RelTool (p1,50.000000,5.000000,15.925560,\Rx:=0.000000,\Ry:=2.040994),vel1,zoneval,Extruder\WObj:=Workobject_1;
MoveL RelTool (p1,52.500000,5.000000,15.429362,\Rx:=0.000000,\Ry:=2.727101),vel1,zoneval,Extruder\WObj:=Workobject_1;
MoveL RelTool (p1,55.000000,5.000000,14.747956,\Rx:=0.000000,\Ry:=3.571964),vel1,zoneval,Extruder\WObj:=Workobject_1;
MoveL RelTool (p1,57.500000,5.000000,13.863713,\Rx:=0.000000,\Ry:=5.085978),vel1,zoneval,Extruder\WObj:=Workobject_1;
MoveL RelTool (p1,60.000000,5.000000,12.681905,\Rx:=0.000000,\Ry:=6.787941),vel1,zoneval,Extruder\WObj:=Workobject_1;
MoveL RelTool (p1,62.500000,5.000000,11.041375,\Rx:=0.000000,\Ry:=8.629267),vel1,zoneval,Extruder\WObj:=Workobject_1;
MoveL RelTool (p1,65.000000,5.000000,8.448953,\Rx:=0.000000,\Ry:=10.686183),vel1,zoneval,Extruder\WObj:=Workobject_1;
MoveL RelTool (p1,67.500000,5.000000,6.722776,\Rx:=0.000000,\Ry:=3.081723),vel1,zoneval,Extruder\WObj:=Workobject_1;
MoveL RelTool (p1,70.000000,5.000000,6.500000,\Rx:=0.000000,\Ry:=-0.000000),vel1,zoneval,Extruder\WObj:=Workobject_1;
MoveL RelTool (p1,72.500000,5.000000,6.500000,\Rx:=0.000000,\Ry:=-0.000000),vel1,zoneval,Extruder\WObj:=Workobject_1;
MoveL RelTool (p1,75.000000,5.000000,6.500000,\Rx:=0.000000,\Ry:=-0.000000),vel1,zoneval,Extruder\WObj:=Workobject_1;
MoveL RelTool (p1,77.500000,5.000000,6.500000,\Rx:=0.000000,\Ry:=-0.000000),vel1,zoneval,Extruder\WObj:=Workobject_1;
MoveL RelTool (p1,80.000000,5.000000,6.500000,\Rx:=0.000000,\Ry:=-0.000000),vel1,zoneval,Extruder\WObj:=Workobject_1;
MoveL RelTool (p1,82.500000,5.000000,6.500000,\Rx:=0.000000,\Ry:=-0.000000),vel1,zoneval,Extruder\WObj:=Workobject_1;
MoveL RelTool (p1,80.500000,5.500000,6.500000,\Rx:=0.000000,\Ry:=0.000000),vel1,zoneval,Extruder\WObj:=Workobject_1;
MoveL RelTool (p1,78.000000,5.500000,6.500000,\Rx:=0.000000,\Ry:=0.000000),vel1,zoneval,Extruder\WObj:=Workobject_1;
MoveL RelTool (p1,75.500000,5.500000,6.500000,\Rx:=0.000000,\Ry:=0.000000),vel1,zoneval,Extruder\WObj:=Workobject_1;
MoveL RelTool (p1,73.000000,5.500000,6.500000,\Rx:=0.000000,\Ry:=0.000000),vel1,zoneval,Extruder\WObj:=Workobject_1;
MoveL RelTool (p1,70.500000,5.500000,6.500000,\Rx:=0.000000,\Ry:=0.000000),vel1,zoneval,Extruder\WObj:=Workobject_1;
MoveL RelTool (p1,68.000000,5.500000,6.599337,\Rx:=0.000000,\Ry:=3.081723),vel1,zoneval,Extruder\WObj:=Workobject_1;
MoveL RelTool (p1,65.500000,5.500000,7.891932,\Rx:=0.000000,\Ry:=10.686183),vel1,zoneval,Extruder\WObj:=Workobject_1;
MoveL RelTool (p1,63.000000,5.500000,10.639954,\Rx:=0.000000,\Ry:=8.619851),vel1,zoneval,Extruder\WObj:=Workobject_1;
MoveL RelTool (p1,60.500000,5.500000,12.387940,\Rx:=0.000000,\Ry:=6.787941),vel1,zoneval,Extruder\WObj:=Workobject_1;
MoveL RelTool (p1,58.000000,5.500000,13.654007,\Rx:=0.000000,\Ry:=5.071511),vel1,zoneval,Extruder\WObj:=Workobject_1;
MoveL RelTool (p1,55.500000,5.500000,14.603622,\Rx:=0.000000,\Ry:=3.578007),vel1,zoneval,Extruder\WObj:=Workobject_1;
MoveL RelTool (p1,53.000000,5.500000,15.320594,\Rx:=0.000000,\Ry:=2.750750),vel1,zoneval,Extruder\WObj:=Workobject_1;
MoveL RelTool (p1,50.500000,5.500000,15.845102,\Rx:=0.000000,\Ry:=2.042981),vel1,zoneval,Extruder\WObj:=Workobject_1;
MoveL RelTool (p1,48.000000,5.500000,16.197648,\Rx:=0.000000,\Ry:=1.667319),vel1,zoneval,Extruder\WObj:=Workobject_1;
MoveL RelTool (p1,45.500000,5.500000,16.406987,\Rx:=0.000000,\Ry:=0.864966),vel1,zoneval,Extruder\WObj:=Workobject_1;
MoveL RelTool (p1,43.000000,5.500000,16.479481,\Rx:=0.000000,\Ry:=0.012935),vel1,zoneval,Extruder\WObj:=Workobject_1;
MoveL RelTool (p1,40.500000,5.500000,16.417502,\Rx:=0.000000,\Ry:=-0.840101),vel1,zoneval,Extruder\WObj:=Workobject_1;
MoveL RelTool (p1,38.000000,5.500000,16.218991,\Rx:=0.000000,\Ry:=-1.705318),vel1,zoneval,Extruder\WObj:=Workobject_1;
MoveL RelTool (p1,35.500000,5.500000,15.875347,\Rx:=0.000000,\Ry:=-2.582835),vel1,zoneval,Extruder\WObj:=Workobject_1;
MoveL RelTool (p1,33.000000,5.500000,15.355168,\Rx:=0.000000,\Ry:=-3.054810),vel1,zoneval,Extruder\WObj:=Workobject_1;
MoveL RelTool (p1,30.500000,5.500000,14.654294,\Rx:=0.000000,\Ry:=-4.128121),vel1,zoneval,Extruder\WObj:=Workobject_1;
MoveL RelTool (p1,28.000000,5.500000,13.731551,\Rx:=0.000000,\Ry:=-5.500143),vel1,zoneval,Extruder\WObj:=Workobject_1;
MoveL RelTool (p1,25.500000,5.500000,12.492763,\Rx:=0.000000,\Ry:=-6.983793),vel1,zoneval,Extruder\WObj:=Workobject_1;
MoveL RelTool (p1,23.000000,5.500000,10.779625,\Rx:=0.000000,\Ry:=-9.254259),vel1,zoneval,Extruder\WObj:=Workobject_1;
MoveL RelTool (p1,20.500000,5.500000,8.040772,\Rx:=0.000000,\Ry:=-9.245074),vel1,zoneval,Extruder\WObj:=Workobject_1;
MoveL RelTool (p1,18.000000,5.500000,6.640720,\Rx:=0.000000,\Ry:=-2.301628),vel1,zoneval,Extruder\WObj:=Workobject_1;
MoveL RelTool (p1,15.500000,5.500000,6.500000,\Rx:=0.000000,\Ry:=0.000000),vel1,zoneval,Extruder\WObj:=Workobject_1;
MoveL RelTool (p1,13.000000,5.500000,6.500000,\Rx:=0.000000,\Ry:=0.000000),vel1,zoneval,Extruder\WObj:=Workobject_1;
MoveL RelTool (p1,10.500000,5.500000,6.500000,\Rx:=0.000000,\Ry:=0.000000),vel1,zoneval,Extruder\WObj:=Workobject_1;
MoveL RelTool (p1,8.000000,5.500000,6.500000,\Rx:=0.000000,\Ry:=0.000000),vel1,zoneval,Extruder\WObj:=Workobject_1;
MoveL RelTool (p1,5.500000,5.500000,6.500000,\Rx:=0.000000,\Ry:=0.000000),vel1,zoneval,Extruder\WObj:=Workobject_1;
MoveL RelTool (p1,3.000000,5.500000,6.500000,\Rx:=0.000000,\Ry:=0.000000),vel1,zoneval,Extruder\WObj:=Workobject_1;
MoveL RelTool (p1,5.000000,6.000000,6.500000,\Rx:=0.000000,\Ry:=-0.000000),vel1,zoneval,Extruder\WObj:=Workobject_1;
MoveL RelTool (p1,7.500000,6.000000,6.500000,\Rx:=0.000000,\Ry:=-0.000000),vel1,zoneval,Extruder\WObj:=Workobject_1;
MoveL RelTool (p1,10.000000,6.000000,6.500000,\Rx:=0.000000,\Ry:=-0.000000),vel1,zoneval,Extruder\WObj:=Workobject_1;
MoveL RelTool (p1,12.500000,6.000000,6.500000,\Rx:=0.000000,\Ry:=-0.000000),vel1,zoneval,Extruder\WObj:=Workobject_1;
MoveL RelTool (p1,15.000000,6.000000,6.500000,\Rx:=0.000000,\Ry:=-0.000000),vel1,zoneval,Extruder\WObj:=Workobject_1;
MoveL RelTool (p1,17.500000,6.000000,6.549338,\Rx:=0.000000,\Ry:=-2.301628),vel1,zoneval,Extruder\WObj:=Workobject_1;
MoveL RelTool (p1,20.000000,6.000000,7.596807,\Rx:=0.000000,\Ry:=-9.245074),vel1,zoneval,Extruder\WObj:=Workobject_1;
MoveL RelTool (p1,22.500000,6.000000,10.335552,\Rx:=0.000000,\Ry:=-9.264444),vel1,zoneval,Extruder\WObj:=Workobject_1;
MoveL RelTool (p1,25.000000,6.000000,12.188371,\Rx:=0.000000,\Ry:=-6.983793),vel1,zoneval,Extruder\WObj:=Workobject_1;
MoveL RelTool (p1,27.500000,6.000000,13.501759,\Rx:=0.000000,\Ry:=-5.478055),vel1,zoneval,Extruder\WObj:=Workobject_1;
MoveL RelTool (p1,30.000000,6.000000,14.486592,\Rx:=0.000000,\Ry:=-4.138904),vel1,zoneval,Extruder\WObj:=Workobject_1;
MoveL RelTool (p1,32.500000,6.000000,15.233132,\Rx:=0.000000,\Ry:=-3.055086),vel1,zoneval,Extruder\WObj:=Workobject_1;
MoveL RelTool (p1,35.000000,6.000000,15.773346,\Rx:=0.000000,\Ry:=-2.554672),vel1,zoneval,Extruder\WObj:=Workobject_1;
MoveL RelTool (p1,37.500000,6.000000,16.152279,\Rx:=0.000000,\Ry:=-1.705318),vel1,zoneval,Extruder\WObj:=Workobject_1;
MoveL RelTool (p1,40.000000,6.000000,16.385365,\Rx:=0.000000,\Ry:=-0.840101),vel1,zoneval,Extruder\WObj:=Workobject_1;
MoveL RelTool (p1,42.500000,6.000000,16.480959,\Rx:=0.000000,\Ry:=0.012935),vel1,zoneval,Extruder\WObj:=Workobject_1;
MoveL RelTool (p1,45.000000,6.000000,16.441834,\Rx:=0.000000,\Ry:=0.864966),vel1,zoneval,Extruder\WObj:=Workobject_1;
MoveL RelTool (p1,47.500000,6.000000,16.263182,\Rx:=0.000000,\Ry:=1.646490),vel1,zoneval,Extruder\WObj:=Workobject_1;
MoveL RelTool (p1,50.000000,6.000000,15.926490,\Rx:=0.000000,\Ry:=2.060517),vel1,zoneval,Extruder\WObj:=Workobject_1;
MoveL RelTool (p1,52.500000,6.000000,15.431295,\Rx:=0.000000,\Ry:=2.774379),vel1,zoneval,Extruder\WObj:=Workobject_1;
MoveL RelTool (p1,55.000000,6.000000,14.749538,\Rx:=0.000000,\Ry:=3.621519),vel1,zoneval,Extruder\WObj:=Workobject_1;
MoveL RelTool (p1,57.500000,6.000000,13.865109,\Rx:=0.000000,\Ry:=5.057030),vel1,zoneval,Extruder\WObj:=Workobject_1;
MoveL RelTool (p1,60.000000,6.000000,12.684096,\Rx:=0.000000,\Ry:=6.787941),vel1,zoneval,Extruder\WObj:=Workobject_1;
MoveL RelTool (p1,62.500000,6.000000,11.042247,\Rx:=0.000000,\Ry:=8.607674),vel1,zoneval,Extruder\WObj:=Workobject_1;
MoveL RelTool (p1,65.000000,6.000000,8.448953,\Rx:=0.000000,\Ry:=10.686183),vel1,zoneval,Extruder\WObj:=Workobject_1;
MoveL RelTool (p1,67.500000,6.000000,6.722776,\Rx:=0.000000,\Ry:=3.081723),vel1,zoneval,Extruder\WObj:=Workobject_1;
MoveL RelTool (p1,70.000000,6.000000,6.500000,\Rx:=0.000000,\Ry:=-0.000000),vel1,zoneval,Extruder\WObj:=Workobject_1;
MoveL RelTool (p1,72.500000,6.000000,6.500000,\Rx:=0.000000,\Ry:=-0.000000),vel1,zoneval,Extruder\WObj:=Workobject_1;
MoveL RelTool (p1,75.000000,6.000000,6.500000,\Rx:=0.000000,\Ry:=-0.000000),vel1,zoneval,Extruder\WObj:=Workobject_1;
MoveL RelTool (p1,77.500000,6.000000,6.500000,\Rx:=0.000000,\Ry:=-0.000000),vel1,zoneval,Extruder\WObj:=Workobject_1;
MoveL RelTool (p1,80.000000,6.000000,6.500000,\Rx:=0.000000,\Ry:=-0.000000),vel1,zoneval,Extruder\WObj:=Workobject_1;
MoveL RelTool (p1,82.500000,6.000000,6.500000,\Rx:=0.000000,\Ry:=-0.000000),vel1,zoneval,Extruder\WObj:=Workobject_1;
MoveL RelTool (p1,80.500000,6.500000,6.500000,\Rx:=0.000000,\Ry:=0.000000),vel1,zoneval,Extruder\WObj:=Workobject_1;
MoveL RelTool (p1,78.000000,6.500000,6.500000,\Rx:=0.000000,\Ry:=0.000000),vel1,zoneval,Extruder\WObj:=Workobject_1;
MoveL RelTool (p1,75.500000,6.500000,6.500000,\Rx:=0.000000,\Ry:=0.000000),vel1,zoneval,Extruder\WObj:=Workobject_1;
MoveL RelTool (p1,73.000000,6.500000,6.500000,\Rx:=0.000000,\Ry:=0.000000),vel1,zoneval,Extruder\WObj:=Workobject_1;
MoveL RelTool (p1,70.500000,6.500000,6.500000,\Rx:=0.000000,\Ry:=0.000000),vel1,zoneval,Extruder\WObj:=Workobject_1;
MoveL RelTool (p1,68.000000,6.500000,6.599337,\Rx:=0.000000,\Ry:=3.081723),vel1,zoneval,Extruder\WObj:=Workobject_1;
MoveL RelTool (p1,65.500000,6.500000,7.891932,\Rx:=0.000000,\Ry:=10.686183),vel1,zoneval,Extruder\WObj:=Workobject_1;
MoveL RelTool (p1,63.000000,6.500000,10.642398,\Rx:=0.000000,\Ry:=8.595970),vel1,zoneval,Extruder\WObj:=Workobject_1;
MoveL RelTool (p1,60.500000,6.500000,12.390131,\Rx:=0.000000,\Ry:=6.787941),vel1,zoneval,Extruder\WObj:=Workobject_1;
MoveL RelTool (p1,58.000000,6.500000,13.656740,\Rx:=0.000000,\Ry:=5.042536),vel1,zoneval,Extruder\WObj:=Workobject_1;
MoveL RelTool (p1,55.500000,6.500000,14.603094,\Rx:=0.000000,\Ry:=3.665822),vel1,zoneval,Extruder\WObj:=Workobject_1;
MoveL RelTool (p1,53.000000,6.500000,15.320581,\Rx:=0.000000,\Ry:=2.797989),vel1,zoneval,Extruder\WObj:=Workobject_1;
MoveL RelTool (p1,50.500000,6.500000,15.844618,\Rx:=0.000000,\Ry:=2.078046),vel1,zoneval,Extruder\WObj:=Workobject_1;
MoveL RelTool (p1,48.000000,6.500000,16.199038,\Rx:=0.000000,\Ry:=1.616560),vel1,zoneval,Extruder\WObj:=Workobject_1;
MoveL RelTool (p1,45.500000,6.500000,16.408642,\Rx:=0.000000,\Ry:=0.861451),vel1,zoneval,Extruder\WObj:=Workobject_1;
MoveL RelTool (p1,43.000000,6.500000,16.481422,\Rx:=0.000000,\Ry:=0.012935),vel1,zoneval,Extruder\WObj:=Workobject_1;
MoveL RelTool (p1,40.500000,6.500000,16.419305,\Rx:=0.000000,\Ry:=-0.840101),vel1,zoneval,Extruder\WObj:=Workobject_1;
MoveL RelTool (p1,38.000000,6.500000,16.220308,\Rx:=0.000000,\Ry:=-1.705318),vel1,zoneval,Extruder\WObj:=Workobject_1;
MoveL RelTool (p1,35.500000,6.500000,15.874725,\Rx:=0.000000,\Ry:=-2.512980),vel1,zoneval,Extruder\WObj:=Workobject_1;
MoveL RelTool (p1,33.000000,6.500000,15.355755,\Rx:=0.000000,\Ry:=-3.065250),vel1,zoneval,Extruder\WObj:=Workobject_1;
MoveL RelTool (p1,30.500000,6.500000,14.654945,\Rx:=0.000000,\Ry:=-4.127521),vel1,zoneval,Extruder\WObj:=Workobject_1;
MoveL RelTool (p1,28.000000,6.500000,13.730885,\Rx:=0.000000,\Ry:=-5.453759),vel1,zoneval,Extruder\WObj:=Workobject_1;
MoveL RelTool (p1,25.500000,6.500000,12.495031,\Rx:=0.000000,\Ry:=-6.983793),vel1,zoneval,Extruder\WObj:=Workobject_1;
MoveL RelTool (p1,23.000000,6.500000,10.782133,\Rx:=0.000000,\Ry:=-9.274615),vel1,zoneval,Extruder\WObj:=Workobject_1;
MoveL RelTool (p1,20.500000,6.500000,8.040772,\Rx:=0.000000,\Ry:=-9.245074),vel1,zoneval,Extruder\WObj:=Workobject_1;
MoveL RelTool (p1,18.000000,6.500000,6.640720,\Rx:=0.000000,\Ry:=-2.301628),vel1,zoneval,Extruder\WObj:=Workobject_1;
MoveL RelTool (p1,15.500000,6.500000,6.500000,\Rx:=0.000000,\Ry:=0.000000),vel1,zoneval,Extruder\WObj:=Workobject_1;
MoveL RelTool (p1,13.000000,6.500000,6.500000,\Rx:=0.000000,\Ry:=0.000000),vel1,zoneval,Extruder\WObj:=Workobject_1;
MoveL RelTool (p1,10.500000,6.500000,6.500000,\Rx:=0.000000,\Ry:=0.000000),vel1,zoneval,Extruder\WObj:=Workobject_1;
MoveL RelTool (p1,8.000000,6.500000,6.500000,\Rx:=0.000000,\Ry:=0.000000),vel1,zoneval,Extruder\WObj:=Workobject_1;
MoveL RelTool (p1,5.500000,6.500000,6.500000,\Rx:=0.000000,\Ry:=0.000000),vel1,zoneval,Extruder\WObj:=Workobject_1;
MoveL RelTool (p1,3.000000,6.500000,6.500000,\Rx:=0.000000,\Ry:=0.000000),vel1,zoneval,Extruder\WObj:=Workobject_1;
MoveL RelTool (p1,5.000000,7.000000,6.500000,\Rx:=0.000000,\Ry:=-0.000000),vel1,zoneval,Extruder\WObj:=Workobject_1;
MoveL RelTool (p1,7.500000,7.000000,6.500000,\Rx:=0.000000,\Ry:=-0.000000),vel1,zoneval,Extruder\WObj:=Workobject_1;
MoveL RelTool (p1,10.000000,7.000000,6.500000,\Rx:=0.000000,\Ry:=-0.000000),vel1,zoneval,Extruder\WObj:=Workobject_1;
MoveL RelTool (p1,12.500000,7.000000,6.500000,\Rx:=0.000000,\Ry:=-0.000000),vel1,zoneval,Extruder\WObj:=Workobject_1;
MoveL RelTool (p1,15.000000,7.000000,6.500000,\Rx:=0.000000,\Ry:=-0.000000),vel1,zoneval,Extruder\WObj:=Workobject_1;
MoveL RelTool (p1,17.500000,7.000000,6.549338,\Rx:=0.000000,\Ry:=-2.301628),vel1,zoneval,Extruder\WObj:=Workobject_1;
MoveL RelTool (p1,20.000000,7.000000,7.596807,\Rx:=0.000000,\Ry:=-9.245074),vel1,zoneval,Extruder\WObj:=Workobject_1;
MoveL RelTool (p1,22.500000,7.000000,10.336627,\Rx:=0.000000,\Ry:=-9.284771),vel1,zoneval,Extruder\WObj:=Workobject_1;
MoveL RelTool (p1,25.000000,7.000000,12.190639,\Rx:=0.000000,\Ry:=-6.983793),vel1,zoneval,Extruder\WObj:=Workobject_1;
MoveL RelTool (p1,27.500000,7.000000,13.503479,\Rx:=0.000000,\Ry:=-5.427761),vel1,zoneval,Extruder\WObj:=Workobject_1;
MoveL RelTool (p1,30.000000,7.000000,14.487269,\Rx:=0.000000,\Ry:=-4.116131),vel1,zoneval,Extruder\WObj:=Workobject_1;
MoveL RelTool (p1,32.500000,7.000000,15.232873,\Rx:=0.000000,\Ry:=-3.075410),vel1,zoneval,Extruder\WObj:=Workobject_1;
MoveL RelTool (p1,35.000000,7.000000,15.776132,\Rx:=0.000000,\Ry:=-2.471233),vel1,zoneval,Extruder\WObj:=Workobject_1;
MoveL RelTool (p1,37.500000,7.000000,16.153596,\Rx:=0.000000,\Ry:=-1.705318),vel1,zoneval,Extruder\WObj:=Workobject_1;
MoveL RelTool (p1,40.000000,7.000000,16.387167,\Rx:=0.000000,\Ry:=-0.840101),vel1,zoneval,Extruder\WObj:=Workobject_1;
MoveL RelTool (p1,42.500000,7.000000,16.482900,\Rx:=0.000000,\Ry:=0.012935),vel1,zoneval,Extruder\WObj:=Workobject_1;
MoveL RelTool (p1,45.000000,7.000000,16.442806,\Rx:=0.000000,\Ry:=0.847667),vel1,zoneval,Extruder\WObj:=Workobject_1;
MoveL RelTool (p1,47.500000,7.000000,16.262545,\Rx:=0.000000,\Ry:=1.586612),vel1,zoneval,Extruder\WObj:=Workobject_1;
MoveL RelTool (p1,50.000000,7.000000,15.927420,\Rx:=0.000000,\Ry:=2.095566),vel1,zoneval,Extruder\WObj:=Workobject_1;
MoveL RelTool (p1,52.500000,7.000000,15.433228,\Rx:=0.000000,\Ry:=2.821579),vel1,zoneval,Extruder\WObj:=Workobject_1;
MoveL RelTool (p1,55.000000,7.000000,14.752792,\Rx:=0.000000,\Ry:=3.710034),vel1,zoneval,Extruder\WObj:=Workobject_1;
MoveL RelTool (p1,57.500000,7.000000,13.866504,\Rx:=0.000000,\Ry:=5.028027),vel1,zoneval,Extruder\WObj:=Workobject_1;
MoveL RelTool (p1,60.000000,7.000000,12.686287,\Rx:=0.000000,\Ry:=6.787941),vel1,zoneval,Extruder\WObj:=Workobject_1;
MoveL RelTool (p1,62.500000,7.000000,11.044025,\Rx:=0.000000,\Ry:=8.597339),vel1,zoneval,Extruder\WObj:=Workobject_1;
MoveL RelTool (p1,65.000000,7.000000,8.448953,\Rx:=0.000000,\Ry:=10.686183),vel1,zoneval,Extruder\WObj:=Workobject_1;
MoveL RelTool (p1,67.500000,7.000000,6.722776,\Rx:=0.000000,\Ry:=3.081723),vel1,zoneval,Extruder\WObj:=Workobject_1;
MoveL RelTool (p1,70.000000,7.000000,6.500000,\Rx:=0.000000,\Ry:=-0.000000),vel1,zoneval,Extruder\WObj:=Workobject_1;
MoveL RelTool (p1,72.500000,7.000000,6.500000,\Rx:=0.000000,\Ry:=-0.000000),vel1,zoneval,Extruder\WObj:=Workobject_1;
MoveL RelTool (p1,75.000000,7.000000,6.500000,\Rx:=0.000000,\Ry:=-0.000000),vel1,zoneval,Extruder\WObj:=Workobject_1;
MoveL RelTool (p1,77.500000,7.000000,6.500000,\Rx:=0.000000,\Ry:=-0.000000),vel1,zoneval,Extruder\WObj:=Workobject_1;
MoveL RelTool (p1,80.000000,7.000000,6.500000,\Rx:=0.000000,\Ry:=-0.000000),vel1,zoneval,Extruder\WObj:=Workobject_1;
MoveL RelTool (p1,82.500000,7.000000,6.500000,\Rx:=0.000000,\Ry:=-0.000000),vel1,zoneval,Extruder\WObj:=Workobject_1;
MoveL RelTool (p1,80.500000,7.500000,6.500000,\Rx:=0.000000,\Ry:=0.000000),vel1,zoneval,Extruder\WObj:=Workobject_1;
MoveL RelTool (p1,78.000000,7.500000,6.500000,\Rx:=0.000000,\Ry:=0.000000),vel1,zoneval,Extruder\WObj:=Workobject_1;
MoveL RelTool (p1,75.500000,7.500000,6.500000,\Rx:=0.000000,\Ry:=0.000000),vel1,zoneval,Extruder\WObj:=Workobject_1;
MoveL RelTool (p1,73.000000,7.500000,6.500000,\Rx:=0.000000,\Ry:=0.000000),vel1,zoneval,Extruder\WObj:=Workobject_1;
MoveL RelTool (p1,70.500000,7.500000,6.500000,\Rx:=0.000000,\Ry:=0.000000),vel1,zoneval,Extruder\WObj:=Workobject_1;
MoveL RelTool (p1,68.000000,7.500000,6.599337,\Rx:=0.000000,\Ry:=3.081723),vel1,zoneval,Extruder\WObj:=Workobject_1;
MoveL RelTool (p1,65.500000,7.500000,7.891932,\Rx:=0.000000,\Ry:=10.686183),vel1,zoneval,Extruder\WObj:=Workobject_1;
MoveL RelTool (p1,63.000000,7.500000,10.644843,\Rx:=0.000000,\Ry:=8.598708),vel1,zoneval,Extruder\WObj:=Workobject_1;
MoveL RelTool (p1,60.500000,7.500000,12.392322,\Rx:=0.000000,\Ry:=6.765291),vel1,zoneval,Extruder\WObj:=Workobject_1;
MoveL RelTool (p1,58.000000,7.500000,13.659177,\Rx:=0.000000,\Ry:=5.019954),vel1,zoneval,Extruder\WObj:=Workobject_1;
MoveL RelTool (p1,55.500000,7.500000,14.602567,\Rx:=0.000000,\Ry:=3.754155),vel1,zoneval,Extruder\WObj:=Workobject_1;
MoveL RelTool (p1,53.000000,7.500000,15.320568,\Rx:=0.000000,\Ry:=2.832149),vel1,zoneval,Extruder\WObj:=Workobject_1;
MoveL RelTool (p1,50.500000,7.500000,15.844135,\Rx:=0.000000,\Ry:=2.113078),vel1,zoneval,Extruder\WObj:=Workobject_1;
MoveL RelTool (p1,48.000000,7.500000,16.200791,\Rx:=0.000000,\Ry:=1.556646),vel1,zoneval,Extruder\WObj:=Workobject_1;
MoveL RelTool (p1,45.500000,7.500000,16.410296,\Rx:=0.000000,\Ry:=0.833881),vel1,zoneval,Extruder\WObj:=Workobject_1;
MoveL RelTool (p1,43.000000,7.500000,16.483363,\Rx:=0.000000,\Ry:=0.012935),vel1,zoneval,Extruder\WObj:=Workobject_1;
MoveL RelTool (p1,40.500000,7.500000,16.421107,\Rx:=0.000000,\Ry:=-0.840101),vel1,zoneval,Extruder\WObj:=Workobject_1;
MoveL RelTool (p1,38.000000,7.500000,16.221625,\Rx:=0.000000,\Ry:=-1.705318),vel1,zoneval,Extruder\WObj:=Workobject_1;
MoveL RelTool (p1,35.500000,7.500000,15.874103,\Rx:=0.000000,\Ry:=-2.429432),vel1,zoneval,Extruder\WObj:=Workobject_1;
MoveL RelTool (p1,33.000000,7.500000,15.356342,\Rx:=0.000000,\Ry:=-3.085566),vel1,zoneval,Extruder\WObj:=Workobject_1;
MoveL RelTool (p1,30.500000,7.500000,14.654627,\Rx:=0.000000,\Ry:=-4.104735),vel1,zoneval,Extruder\WObj:=Workobject_1;
MoveL RelTool (p1,28.000000,7.500000,13.730219,\Rx:=0.000000,\Ry:=-5.401715),vel1,zoneval,Extruder\WObj:=Workobject_1;
MoveL RelTool (p1,25.500000,7.500000,12.497299,\Rx:=0.000000,\Ry:=-6.983793),vel1,zoneval,Extruder\WObj:=Workobject_1;
MoveL RelTool (p1,23.000000,7.500000,10.784642,\Rx:=0.000000,\Ry:=-9.294913),vel1,zoneval,Extruder\WObj:=Workobject_1;
MoveL RelTool (p1,20.500000,7.500000,8.040772,\Rx:=0.000000,\Ry:=-9.245074),vel1,zoneval,Extruder\WObj:=Workobject_1;
MoveL RelTool (p1,18.000000,7.500000,6.640720,\Rx:=0.000000,\Ry:=-2.301628),vel1,zoneval,Extruder\WObj:=Workobject_1;
MoveL RelTool (p1,15.500000,7.500000,6.500000,\Rx:=0.000000,\Ry:=0.000000),vel1,zoneval,Extruder\WObj:=Workobject_1;
MoveL RelTool (p1,13.000000,7.500000,6.500000,\Rx:=0.000000,\Ry:=0.000000),vel1,zoneval,Extruder\WObj:=Workobject_1;
MoveL RelTool (p1,10.500000,7.500000,6.500000,\Rx:=0.000000,\Ry:=0.000000),vel1,zoneval,Extruder\WObj:=Workobject_1;
MoveL RelTool (p1,8.000000,7.500000,6.500000,\Rx:=0.000000,\Ry:=0.000000),vel1,zoneval,Extruder\WObj:=Workobject_1;
MoveL RelTool (p1,5.500000,7.500000,6.500000,\Rx:=0.000000,\Ry:=0.000000),vel1,zoneval,Extruder\WObj:=Workobject_1;
MoveL RelTool (p1,3.000000,7.500000,6.500000,\Rx:=0.000000,\Ry:=0.000000),vel1,zoneval,Extruder\WObj:=Workobject_1;
MoveL RelTool (p1,5.000000,8.000000,6.500000,\Rx:=0.000000,\Ry:=-0.000000),vel1,zoneval,Extruder\WObj:=Workobject_1;
MoveL RelTool (p1,7.500000,8.000000,6.500000,\Rx:=0.000000,\Ry:=-0.000000),vel1,zoneval,Extruder\WObj:=Workobject_1;
MoveL RelTool (p1,10.000000,8.000000,6.500000,\Rx:=0.000000,\Ry:=-0.000000),vel1,zoneval,Extruder\WObj:=Workobject_1;
MoveL RelTool (p1,12.500000,8.000000,6.500000,\Rx:=0.000000,\Ry:=-0.000000),vel1,zoneval,Extruder\WObj:=Workobject_1;
MoveL RelTool (p1,15.000000,8.000000,6.500000,\Rx:=0.000000,\Ry:=-0.000000),vel1,zoneval,Extruder\WObj:=Workobject_1;
MoveL RelTool (p1,17.500000,8.000000,6.549338,\Rx:=0.000000,\Ry:=-2.301628),vel1,zoneval,Extruder\WObj:=Workobject_1;
MoveL RelTool (p1,20.000000,8.000000,7.596807,\Rx:=0.000000,\Ry:=-9.245074),vel1,zoneval,Extruder\WObj:=Workobject_1;
MoveL RelTool (p1,22.500000,8.000000,10.337702,\Rx:=0.000000,\Ry:=-9.305040),vel1,zoneval,Extruder\WObj:=Workobject_1;
MoveL RelTool (p1,25.000000,8.000000,12.192907,\Rx:=0.000000,\Ry:=-6.983793),vel1,zoneval,Extruder\WObj:=Workobject_1;
MoveL RelTool (p1,27.500000,8.000000,13.505279,\Rx:=0.000000,\Ry:=-5.375621),vel1,zoneval,Extruder\WObj:=Workobject_1;
MoveL RelTool (p1,30.000000,8.000000,14.487947,\Rx:=0.000000,\Ry:=-4.093331),vel1,zoneval,Extruder\WObj:=Workobject_1;
MoveL RelTool (p1,32.500000,8.000000,15.232613,\Rx:=0.000000,\Ry:=-3.095718),vel1,zoneval,Extruder\WObj:=Workobject_1;
MoveL RelTool (p1,35.000000,8.000000,15.778917,\Rx:=0.000000,\Ry:=-2.387578),vel1,zoneval,Extruder\WObj:=Workobject_1;
MoveL RelTool (p1,37.500000,8.000000,16.154913,\Rx:=0.000000,\Ry:=-1.705318),vel1,zoneval,Extruder\WObj:=Workobject_1;
MoveL RelTool (p1,40.000000,8.000000,16.388970,\Rx:=0.000000,\Ry:=-0.840101),vel1,zoneval,Extruder\WObj:=Workobject_1;
MoveL RelTool (p1,42.500000,8.000000,16.484842,\Rx:=0.000000,\Ry:=0.012935),vel1,zoneval,Extruder\WObj:=Workobject_1;
MoveL RelTool (p1,45.000000,8.000000,16.443373,\Rx:=0.000000,\Ry:=0.820093),vel1,zoneval,Extruder\WObj:=Workobject_1;
MoveL RelTool (p1,47.500000,8.000000,16.261909,\Rx:=0.000000,\Ry:=1.526663),vel1,zoneval,Extruder\WObj:=Workobject_1;
MoveL RelTool (p1,50.000000,8.000000,15.928351,\Rx:=0.000000,\Ry:=2.130583),vel1,zoneval,Extruder\WObj:=Workobject_1;
MoveL RelTool (p1,52.500000,8.000000,15.433651,\Rx:=0.000000,\Ry:=2.832151),vel1,zoneval,Extruder\WObj:=Workobject_1;
MoveL RelTool (p1,55.000000,8.000000,14.756045,\Rx:=0.000000,\Ry:=3.798182),vel1,zoneval,Extruder\WObj:=Workobject_1;
MoveL RelTool (p1,57.500000,8.000000,13.867900,\Rx:=0.000000,\Ry:=5.041964),vel1,zoneval,Extruder\WObj:=Workobject_1;
MoveL RelTool (p1,60.000000,8.000000,12.686039,\Rx:=0.000000,\Ry:=6.741768),vel1,zoneval,Extruder\WObj:=Workobject_1;
MoveL RelTool (p1,62.500000,8.000000,11.046645,\Rx:=0.000000,\Ry:=8.600077),vel1,zoneval,Extruder\WObj:=Workobject_1;
MoveL RelTool (p1,65.000000,8.000000,8.448953,\Rx:=0.000000,\Ry:=10.686183),vel1,zoneval,Extruder\WObj:=Workobject_1;
MoveL RelTool (p1,67.500000,8.000000,6.722776,\Rx:=0.000000,\Ry:=3.081723),vel1,zoneval,Extruder\WObj:=Workobject_1;
MoveL RelTool (p1,70.000000,8.000000,6.500000,\Rx:=0.000000,\Ry:=-0.000000),vel1,zoneval,Extruder\WObj:=Workobject_1;
MoveL RelTool (p1,72.500000,8.000000,6.500000,\Rx:=0.000000,\Ry:=-0.000000),vel1,zoneval,Extruder\WObj:=Workobject_1;
MoveL RelTool (p1,75.000000,8.000000,6.500000,\Rx:=0.000000,\Ry:=-0.000000),vel1,zoneval,Extruder\WObj:=Workobject_1;
MoveL RelTool (p1,77.500000,8.000000,6.500000,\Rx:=0.000000,\Ry:=-0.000000),vel1,zoneval,Extruder\WObj:=Workobject_1;
MoveL RelTool (p1,80.000000,8.000000,6.500000,\Rx:=0.000000,\Ry:=-0.000000),vel1,zoneval,Extruder\WObj:=Workobject_1;
MoveL RelTool (p1,82.500000,8.000000,6.500000,\Rx:=0.000000,\Ry:=-0.000000),vel1,zoneval,Extruder\WObj:=Workobject_1;
MoveL RelTool (p1,80.500000,8.500000,6.500000,\Rx:=0.000000,\Ry:=0.000000),vel1,zoneval,Extruder\WObj:=Workobject_1;
MoveL RelTool (p1,78.000000,8.500000,6.500000,\Rx:=0.000000,\Ry:=0.000000),vel1,zoneval,Extruder\WObj:=Workobject_1;
MoveL RelTool (p1,75.500000,8.500000,6.500000,\Rx:=0.000000,\Ry:=0.000000),vel1,zoneval,Extruder\WObj:=Workobject_1;
MoveL RelTool (p1,73.000000,8.500000,6.500000,\Rx:=0.000000,\Ry:=0.000000),vel1,zoneval,Extruder\WObj:=Workobject_1;
MoveL RelTool (p1,70.500000,8.500000,6.500000,\Rx:=0.000000,\Ry:=0.000000),vel1,zoneval,Extruder\WObj:=Workobject_1;
MoveL RelTool (p1,68.000000,8.500000,6.599337,\Rx:=0.000000,\Ry:=3.081723),vel1,zoneval,Extruder\WObj:=Workobject_1;
MoveL RelTool (p1,65.500000,8.500000,7.891932,\Rx:=0.000000,\Ry:=10.686183),vel1,zoneval,Extruder\WObj:=Workobject_1;
MoveL RelTool (p1,63.000000,8.500000,10.647287,\Rx:=0.000000,\Ry:=8.601446),vel1,zoneval,Extruder\WObj:=Workobject_1;
MoveL RelTool (p1,60.500000,8.500000,12.394514,\Rx:=0.000000,\Ry:=6.718194),vel1,zoneval,Extruder\WObj:=Workobject_1;
MoveL RelTool (p1,58.000000,8.500000,13.658543,\Rx:=0.000000,\Ry:=5.063942),vel1,zoneval,Extruder\WObj:=Workobject_1;
MoveL RelTool (p1,55.500000,8.500000,14.602040,\Rx:=0.000000,\Ry:=3.842117),vel1,zoneval,Extruder\WObj:=Workobject_1;
MoveL RelTool (p1,53.000000,8.500000,15.320554,\Rx:=0.000000,\Ry:=2.832153),vel1,zoneval,Extruder\WObj:=Workobject_1;
MoveL RelTool (p1,50.500000,8.500000,15.843651,\Rx:=0.000000,\Ry:=2.148079),vel1,zoneval,Extruder\WObj:=Workobject_1;
MoveL RelTool (p1,48.000000,8.500000,16.202544,\Rx:=0.000000,\Ry:=1.496663),vel1,zoneval,Extruder\WObj:=Workobject_1;
MoveL RelTool (p1,45.500000,8.500000,16.411951,\Rx:=0.000000,\Ry:=0.806303),vel1,zoneval,Extruder\WObj:=Workobject_1;
MoveL RelTool (p1,43.000000,8.500000,16.485304,\Rx:=0.000000,\Ry:=0.012935),vel1,zoneval,Extruder\WObj:=Workobject_1;
MoveL RelTool (p1,40.500000,8.500000,16.422910,\Rx:=0.000000,\Ry:=-0.840101),vel1,zoneval,Extruder\WObj:=Workobject_1;
MoveL RelTool (p1,38.000000,8.500000,16.222942,\Rx:=0.000000,\Ry:=-1.705318),vel1,zoneval,Extruder\WObj:=Workobject_1;
MoveL RelTool (p1,35.500000,8.500000,15.873481,\Rx:=0.000000,\Ry:=-2.345672),vel1,zoneval,Extruder\WObj:=Workobject_1;
MoveL RelTool (p1,33.000000,8.500000,15.356929,\Rx:=0.000000,\Ry:=-3.105866),vel1,zoneval,Extruder\WObj:=Workobject_1;
MoveL RelTool (p1,30.500000,8.500000,14.654309,\Rx:=0.000000,\Ry:=-4.081921),vel1,zoneval,Extruder\WObj:=Workobject_1;
MoveL RelTool (p1,28.000000,8.500000,13.729553,\Rx:=0.000000,\Ry:=-5.349479),vel1,zoneval,Extruder\WObj:=Workobject_1;
MoveL RelTool (p1,25.500000,8.500000,12.499567,\Rx:=0.000000,\Ry:=-6.983793),vel1,zoneval,Extruder\WObj:=Workobject_1;
MoveL RelTool (p1,23.000000,8.500000,10.786476,\Rx:=0.000000,\Ry:=-9.305645),vel1,zoneval,Extruder\WObj:=Workobject_1;
MoveL RelTool (p1,20.500000,8.500000,8.040772,\Rx:=0.000000,\Ry:=-9.245074),vel1,zoneval,Extruder\WObj:=Workobject_1;
MoveL RelTool (p1,18.000000,8.500000,6.640720,\Rx:=0.000000,\Ry:=-2.301628),vel1,zoneval,Extruder\WObj:=Workobject_1;
MoveL RelTool (p1,15.500000,8.500000,6.500000,\Rx:=0.000000,\Ry:=0.000000),vel1,zoneval,Extruder\WObj:=Workobject_1;
MoveL RelTool (p1,13.000000,8.500000,6.500000,\Rx:=0.000000,\Ry:=0.000000),vel1,zoneval,Extruder\WObj:=Workobject_1;
MoveL RelTool (p1,10.500000,8.500000,6.500000,\Rx:=0.000000,\Ry:=0.000000),vel1,zoneval,Extruder\WObj:=Workobject_1;
MoveL RelTool (p1,8.000000,8.500000,6.500000,\Rx:=0.000000,\Ry:=0.000000),vel1,zoneval,Extruder\WObj:=Workobject_1;
MoveL RelTool (p1,5.500000,8.500000,6.500000,\Rx:=0.000000,\Ry:=0.000000),vel1,zoneval,Extruder\WObj:=Workobject_1;
MoveL RelTool (p1,3.000000,8.500000,6.500000,\Rx:=0.000000,\Ry:=0.000000),vel1,zoneval,Extruder\WObj:=Workobject_1;
MoveL RelTool (p1,5.000000,9.000000,6.500000,\Rx:=0.000000,\Ry:=-0.000000),vel1,zoneval,Extruder\WObj:=Workobject_1;
MoveL RelTool (p1,7.500000,9.000000,6.500000,\Rx:=0.000000,\Ry:=-0.000000),vel1,zoneval,Extruder\WObj:=Workobject_1;
MoveL RelTool (p1,10.000000,9.000000,6.500000,\Rx:=0.000000,\Ry:=-0.000000),vel1,zoneval,Extruder\WObj:=Workobject_1;
MoveL RelTool (p1,12.500000,9.000000,6.500000,\Rx:=0.000000,\Ry:=-0.000000),vel1,zoneval,Extruder\WObj:=Workobject_1;
MoveL RelTool (p1,15.000000,9.000000,6.500000,\Rx:=0.000000,\Ry:=-0.000000),vel1,zoneval,Extruder\WObj:=Workobject_1;
MoveL RelTool (p1,17.500000,9.000000,6.549338,\Rx:=0.000000,\Ry:=-2.301628),vel1,zoneval,Extruder\WObj:=Workobject_1;
MoveL RelTool (p1,20.000000,9.000000,7.596807,\Rx:=0.000000,\Ry:=-9.245074),vel1,zoneval,Extruder\WObj:=Workobject_1;
MoveL RelTool (p1,22.500000,9.000000,10.338776,\Rx:=0.000000,\Ry:=-9.294486),vel1,zoneval,Extruder\WObj:=Workobject_1;
MoveL RelTool (p1,25.000000,9.000000,12.195175,\Rx:=0.000000,\Ry:=-6.983793),vel1,zoneval,Extruder\WObj:=Workobject_1;
MoveL RelTool (p1,27.500000,9.000000,13.507078,\Rx:=0.000000,\Ry:=-5.323288),vel1,zoneval,Extruder\WObj:=Workobject_1;
MoveL RelTool (p1,30.000000,9.000000,14.488624,\Rx:=0.000000,\Ry:=-4.070504),vel1,zoneval,Extruder\WObj:=Workobject_1;
MoveL RelTool (p1,32.500000,9.000000,15.232354,\Rx:=0.000000,\Ry:=-3.116009),vel1,zoneval,Extruder\WObj:=Workobject_1;
MoveL RelTool (p1,35.000000,9.000000,15.781703,\Rx:=0.000000,\Ry:=-2.303714),vel1,zoneval,Extruder\WObj:=Workobject_1;
MoveL RelTool (p1,37.500000,9.000000,16.156230,\Rx:=0.000000,\Ry:=-1.705318),vel1,zoneval,Extruder\WObj:=Workobject_1;
MoveL RelTool (p1,40.000000,9.000000,16.390772,\Rx:=0.000000,\Ry:=-0.840101),vel1,zoneval,Extruder\WObj:=Workobject_1;
MoveL RelTool (p1,42.500000,9.000000,16.486783,\Rx:=0.000000,\Ry:=0.012935),vel1,zoneval,Extruder\WObj:=Workobject_1;
MoveL RelTool (p1,45.000000,9.000000,16.443940,\Rx:=0.000000,\Ry:=0.792512),vel1,zoneval,Extruder\WObj:=Workobject_1;
MoveL RelTool (p1,47.500000,9.000000,16.261272,\Rx:=0.000000,\Ry:=1.466646),vel1,zoneval,Extruder\WObj:=Workobject_1;
MoveL RelTool (p1,50.000000,9.000000,15.929281,\Rx:=0.000000,\Ry:=2.165567),vel1,zoneval,Extruder\WObj:=Workobject_1;
MoveL RelTool (p1,52.500000,9.000000,15.433638,\Rx:=0.000000,\Ry:=2.832155),vel1,zoneval,Extruder\WObj:=Workobject_1;
MoveL RelTool (p1,55.000000,9.000000,14.759299,\Rx:=0.000000,\Ry:=3.885957),vel1,zoneval,Extruder\WObj:=Workobject_1;
MoveL RelTool (p1,57.500000,9.000000,13.869295,\Rx:=0.000000,\Ry:=5.085888),vel1,zoneval,Extruder\WObj:=Workobject_1;
MoveL RelTool (p1,60.000000,9.000000,12.685747,\Rx:=0.000000,\Ry:=6.694570),vel1,zoneval,Extruder\WObj:=Workobject_1;
MoveL RelTool (p1,62.500000,9.000000,11.049266,\Rx:=0.000000,\Ry:=8.602815),vel1,zoneval,Extruder\WObj:=Workobject_1;
MoveL RelTool (p1,65.000000,9.000000,8.448953,\Rx:=0.000000,\Ry:=10.686183),vel1,zoneval,Extruder\WObj:=Workobject_1;
MoveL RelTool (p1,67.500000,9.000000,6.722776,\Rx:=0.000000,\Ry:=3.081723),vel1,zoneval,Extruder\WObj:=Workobject_1;
MoveL RelTool (p1,70.000000,9.000000,6.500000,\Rx:=0.000000,\Ry:=-0.000000),vel1,zoneval,Extruder\WObj:=Workobject_1;
MoveL RelTool (p1,72.500000,9.000000,6.500000,\Rx:=0.000000,\Ry:=-0.000000),vel1,zoneval,Extruder\WObj:=Workobject_1;
MoveL RelTool (p1,75.000000,9.000000,6.500000,\Rx:=0.000000,\Ry:=-0.000000),vel1,zoneval,Extruder\WObj:=Workobject_1;
MoveL RelTool (p1,77.500000,9.000000,6.500000,\Rx:=0.000000,\Ry:=-0.000000),vel1,zoneval,Extruder\WObj:=Workobject_1;
MoveL RelTool (p1,80.000000,9.000000,6.500000,\Rx:=0.000000,\Ry:=-0.000000),vel1,zoneval,Extruder\WObj:=Workobject_1;
MoveL RelTool (p1,82.500000,9.000000,6.500000,\Rx:=0.000000,\Ry:=-0.000000),vel1,zoneval,Extruder\WObj:=Workobject_1;
MoveL RelTool (p1,80.500000,9.500000,6.500000,\Rx:=0.000000,\Ry:=0.000000),vel1,zoneval,Extruder\WObj:=Workobject_1;
MoveL RelTool (p1,78.000000,9.500000,6.500000,\Rx:=0.000000,\Ry:=0.000000),vel1,zoneval,Extruder\WObj:=Workobject_1;
MoveL RelTool (p1,75.500000,9.500000,6.500000,\Rx:=0.000000,\Ry:=0.000000),vel1,zoneval,Extruder\WObj:=Workobject_1;
MoveL RelTool (p1,73.000000,9.500000,6.500000,\Rx:=0.000000,\Ry:=0.000000),vel1,zoneval,Extruder\WObj:=Workobject_1;
MoveL RelTool (p1,70.500000,9.500000,6.500000,\Rx:=0.000000,\Ry:=0.000000),vel1,zoneval,Extruder\WObj:=Workobject_1;
MoveL RelTool (p1,68.000000,9.500000,6.599337,\Rx:=0.000000,\Ry:=3.081723),vel1,zoneval,Extruder\WObj:=Workobject_1;
MoveL RelTool (p1,65.500000,9.500000,7.891932,\Rx:=0.000000,\Ry:=10.686183),vel1,zoneval,Extruder\WObj:=Workobject_1;
MoveL RelTool (p1,63.000000,9.500000,10.649590,\Rx:=0.000000,\Ry:=8.606377),vel1,zoneval,Extruder\WObj:=Workobject_1;
MoveL RelTool (p1,60.500000,9.500000,12.396705,\Rx:=0.000000,\Ry:=6.670894),vel1,zoneval,Extruder\WObj:=Workobject_1;
MoveL RelTool (p1,58.000000,9.500000,13.657909,\Rx:=0.000000,\Ry:=5.107803),vel1,zoneval,Extruder\WObj:=Workobject_1;
MoveL RelTool (p1,55.500000,9.500000,14.601512,\Rx:=0.000000,\Ry:=3.924353),vel1,zoneval,Extruder\WObj:=Workobject_1;
MoveL RelTool (p1,53.000000,9.500000,15.320541,\Rx:=0.000000,\Ry:=2.832157),vel1,zoneval,Extruder\WObj:=Workobject_1;
MoveL RelTool (p1,50.500000,9.500000,15.843168,\Rx:=0.000000,\Ry:=2.183046),vel1,zoneval,Extruder\WObj:=Workobject_1;
MoveL RelTool (p1,48.000000,9.500000,16.204298,\Rx:=0.000000,\Ry:=1.436612),vel1,zoneval,Extruder\WObj:=Workobject_1;
MoveL RelTool (p1,45.500000,9.500000,16.413605,\Rx:=0.000000,\Ry:=0.778718),vel1,zoneval,Extruder\WObj:=Workobject_1;
MoveL RelTool (p1,43.000000,9.500000,16.487245,\Rx:=0.000000,\Ry:=0.012935),vel1,zoneval,Extruder\WObj:=Workobject_1;
MoveL RelTool (p1,40.500000,9.500000,16.424712,\Rx:=0.000000,\Ry:=-0.840101),vel1,zoneval,Extruder\WObj:=Workobject_1;
MoveL RelTool (p1,38.000000,9.500000,16.224259,\Rx:=0.000000,\Ry:=-1.705318),vel1,zoneval,Extruder\WObj:=Workobject_1;
MoveL RelTool (p1,35.500000,9.500000,15.872859,\Rx:=0.000000,\Ry:=-2.261706),vel1,zoneval,Extruder\WObj:=Workobject_1;
MoveL RelTool (p1,33.000000,9.500000,15.357516,\Rx:=0.000000,\Ry:=-3.126149),vel1,zoneval,Extruder\WObj:=Workobject_1;
MoveL RelTool (p1,30.500000,9.500000,14.653991,\Rx:=0.000000,\Ry:=-4.059080),vel1,zoneval,Extruder\WObj:=Workobject_1;
MoveL RelTool (p1,28.000000,9.500000,13.728887,\Rx:=0.000000,\Ry:=-5.297050),vel1,zoneval,Extruder\WObj:=Workobject_1;
MoveL RelTool (p1,25.500000,9.500000,12.501835,\Rx:=0.000000,\Ry:=-6.983793),vel1,zoneval,Extruder\WObj:=Workobject_1;
MoveL RelTool (p1,23.000000,9.500000,10.785971,\Rx:=0.000000,\Ry:=-9.283310),vel1,zoneval,Extruder\WObj:=Workobject_1;
MoveL RelTool (p1,20.500000,9.500000,8.040772,\Rx:=0.000000,\Ry:=-9.245074),vel1,zoneval,Extruder\WObj:=Workobject_1;
MoveL RelTool (p1,18.000000,9.500000,6.640720,\Rx:=0.000000,\Ry:=-2.301628),vel1,zoneval,Extruder\WObj:=Workobject_1;
MoveL RelTool (p1,15.500000,9.500000,6.500000,\Rx:=0.000000,\Ry:=0.000000),vel1,zoneval,Extruder\WObj:=Workobject_1;
MoveL RelTool (p1,13.000000,9.500000,6.500000,\Rx:=0.000000,\Ry:=0.000000),vel1,zoneval,Extruder\WObj:=Workobject_1;
MoveL RelTool (p1,10.500000,9.500000,6.500000,\Rx:=0.000000,\Ry:=0.000000),vel1,zoneval,Extruder\WObj:=Workobject_1;
MoveL RelTool (p1,8.000000,9.500000,6.500000,\Rx:=0.000000,\Ry:=0.000000),vel1,zoneval,Extruder\WObj:=Workobject_1;
MoveL RelTool (p1,5.500000,9.500000,6.500000,\Rx:=0.000000,\Ry:=0.000000),vel1,zoneval,Extruder\WObj:=Workobject_1;
MoveL RelTool (p1,3.000000,9.500000,6.500000,\Rx:=0.000000,\Ry:=0.000000),vel1,zoneval,Extruder\WObj:=Workobject_1;
MoveL RelTool (p1,5.000000,10.000000,6.500000,\Rx:=0.000000,\Ry:=-0.000000),vel1,zoneval,Extruder\WObj:=Workobject_1;
MoveL RelTool (p1,7.500000,10.000000,6.500000,\Rx:=0.000000,\Ry:=-0.000000),vel1,zoneval,Extruder\WObj:=Workobject_1;
MoveL RelTool (p1,10.000000,10.000000,6.500000,\Rx:=0.000000,\Ry:=-0.000000),vel1,zoneval,Extruder\WObj:=Workobject_1;
MoveL RelTool (p1,12.500000,10.000000,6.500000,\Rx:=0.000000,\Ry:=-0.000000),vel1,zoneval,Extruder\WObj:=Workobject_1;
MoveL RelTool (p1,15.000000,10.000000,6.500000,\Rx:=0.000000,\Ry:=-0.000000),vel1,zoneval,Extruder\WObj:=Workobject_1;
MoveL RelTool (p1,17.500000,10.000000,6.549338,\Rx:=0.000000,\Ry:=-2.301628),vel1,zoneval,Extruder\WObj:=Workobject_1;
MoveL RelTool (p1,20.000000,10.000000,7.596807,\Rx:=0.000000,\Ry:=-9.245074),vel1,zoneval,Extruder\WObj:=Workobject_1;
MoveL RelTool (p1,22.500000,10.000000,10.339851,\Rx:=0.000000,\Ry:=-9.272116),vel1,zoneval,Extruder\WObj:=Workobject_1;
MoveL RelTool (p1,25.000000,10.000000,12.197443,\Rx:=0.000000,\Ry:=-6.974470),vel1,zoneval,Extruder\WObj:=Workobject_1;
MoveL RelTool (p1,27.500000,10.000000,13.508877,\Rx:=0.000000,\Ry:=-5.270764),vel1,zoneval,Extruder\WObj:=Workobject_1;
MoveL RelTool (p1,30.000000,10.000000,14.489301,\Rx:=0.000000,\Ry:=-4.047649),vel1,zoneval,Extruder\WObj:=Workobject_1;
MoveL RelTool (p1,32.500000,10.000000,15.232095,\Rx:=0.000000,\Ry:=-3.136285),vel1,zoneval,Extruder\WObj:=Workobject_1;
MoveL RelTool (p1,35.000000,10.000000,15.784489,\Rx:=0.000000,\Ry:=-2.219647),vel1,zoneval,Extruder\WObj:=Workobject_1;
MoveL RelTool (p1,37.500000,10.000000,16.157547,\Rx:=0.000000,\Ry:=-1.705318),vel1,zoneval,Extruder\WObj:=Workobject_1;
MoveL RelTool (p1,40.000000,10.000000,16.392575,\Rx:=0.000000,\Ry:=-0.823557),vel1,zoneval,Extruder\WObj:=Workobject_1;
MoveL RelTool (p1,42.500000,10.000000,16.488724,\Rx:=0.000000,\Ry:=0.012935),vel1,zoneval,Extruder\WObj:=Workobject_1;
MoveL RelTool (p1,45.000000,10.000000,16.444507,\Rx:=0.000000,\Ry:=0.777724),vel1,zoneval,Extruder\WObj:=Workobject_1;
MoveL RelTool (p1,47.500000,10.000000,16.260636,\Rx:=0.000000,\Ry:=1.406563),vel1,zoneval,Extruder\WObj:=Workobject_1;
MoveL RelTool (p1,50.000000,10.000000,15.930211,\Rx:=0.000000,\Ry:=2.200518),vel1,zoneval,Extruder\WObj:=Workobject_1;
MoveL RelTool (p1,52.500000,10.000000,15.433625,\Rx:=0.000000,\Ry:=2.832159),vel1,zoneval,Extruder\WObj:=Workobject_1;
MoveL RelTool (p1,55.000000,10.000000,14.760431,\Rx:=0.000000,\Ry:=3.924353),vel1,zoneval,Extruder\WObj:=Workobject_1;
MoveL RelTool (p1,57.500000,10.000000,13.869957,\Rx:=0.000000,\Ry:=5.113869),vel1,zoneval,Extruder\WObj:=Workobject_1;
MoveL RelTool (p1,60.000000,10.000000,12.685456,\Rx:=0.000000,\Ry:=6.647168),vel1,zoneval,Extruder\WObj:=Workobject_1;
MoveL RelTool (p1,62.500000,10.000000,11.051887,\Rx:=0.000000,\Ry:=8.632933),vel1,zoneval,Extruder\WObj:=Workobject_1;
MoveL RelTool (p1,65.000000,10.000000,8.448953,\Rx:=0.000000,\Ry:=10.686183),vel1,zoneval,Extruder\WObj:=Workobject_1;
MoveL RelTool (p1,67.500000,10.000000,6.722776,\Rx:=0.000000,\Ry:=3.081723),vel1,zoneval,Extruder\WObj:=Workobject_1;
MoveL RelTool (p1,70.000000,10.000000,6.500000,\Rx:=0.000000,\Ry:=-0.000000),vel1,zoneval,Extruder\WObj:=Workobject_1;
MoveL RelTool (p1,72.500000,10.000000,6.500000,\Rx:=0.000000,\Ry:=-0.000000),vel1,zoneval,Extruder\WObj:=Workobject_1;
MoveL RelTool (p1,75.000000,10.000000,6.500000,\Rx:=0.000000,\Ry:=-0.000000),vel1,zoneval,Extruder\WObj:=Workobject_1;
MoveL RelTool (p1,77.500000,10.000000,6.500000,\Rx:=0.000000,\Ry:=-0.000000),vel1,zoneval,Extruder\WObj:=Workobject_1;
MoveL RelTool (p1,80.000000,10.000000,6.500000,\Rx:=0.000000,\Ry:=-0.000000),vel1,zoneval,Extruder\WObj:=Workobject_1;
MoveL RelTool (p1,82.500000,10.000000,6.500000,\Rx:=0.000000,\Ry:=-0.000000),vel1,zoneval,Extruder\WObj:=Workobject_1;
MoveL RelTool (p1,80.500000,10.500000,6.500000,\Rx:=0.000000,\Ry:=0.000000),vel1,zoneval,Extruder\WObj:=Workobject_1;
MoveL RelTool (p1,78.000000,10.500000,6.500000,\Rx:=0.000000,\Ry:=0.000000),vel1,zoneval,Extruder\WObj:=Workobject_1;
MoveL RelTool (p1,75.500000,10.500000,6.500000,\Rx:=0.000000,\Ry:=0.000000),vel1,zoneval,Extruder\WObj:=Workobject_1;
MoveL RelTool (p1,73.000000,10.500000,6.500000,\Rx:=0.000000,\Ry:=0.000000),vel1,zoneval,Extruder\WObj:=Workobject_1;
MoveL RelTool (p1,70.500000,10.500000,6.500000,\Rx:=0.000000,\Ry:=0.000000),vel1,zoneval,Extruder\WObj:=Workobject_1;
MoveL RelTool (p1,68.000000,10.500000,6.599337,\Rx:=0.000000,\Ry:=3.081723),vel1,zoneval,Extruder\WObj:=Workobject_1;
MoveL RelTool (p1,65.500000,10.500000,7.891932,\Rx:=0.000000,\Ry:=10.686183),vel1,zoneval,Extruder\WObj:=Workobject_1;
MoveL RelTool (p1,63.000000,10.500000,10.648778,\Rx:=0.000000,\Ry:=8.659400),vel1,zoneval,Extruder\WObj:=Workobject_1;
MoveL RelTool (p1,60.500000,10.500000,12.398896,\Rx:=0.000000,\Ry:=6.623390),vel1,zoneval,Extruder\WObj:=Workobject_1;
MoveL RelTool (p1,58.000000,10.500000,13.657275,\Rx:=0.000000,\Ry:=5.113869),vel1,zoneval,Extruder\WObj:=Workobject_1;
MoveL RelTool (p1,55.500000,10.500000,14.600985,\Rx:=0.000000,\Ry:=3.924353),vel1,zoneval,Extruder\WObj:=Workobject_1;
MoveL RelTool (p1,53.000000,10.500000,15.320528,\Rx:=0.000000,\Ry:=2.832161),vel1,zoneval,Extruder\WObj:=Workobject_1;
MoveL RelTool (p1,50.500000,10.500000,15.842684,\Rx:=0.000000,\Ry:=2.217981),vel1,zoneval,Extruder\WObj:=Workobject_1;
MoveL RelTool (p1,48.000000,10.500000,16.206051,\Rx:=0.000000,\Ry:=1.376498),vel1,zoneval,Extruder\WObj:=Workobject_1;
MoveL RelTool (p1,45.500000,10.500000,16.414211,\Rx:=0.000000,\Ry:=0.777724),vel1,zoneval,Extruder\WObj:=Workobject_1;
MoveL RelTool (p1,43.000000,10.500000,16.489186,\Rx:=0.000000,\Ry:=0.012935),vel1,zoneval,Extruder\WObj:=Workobject_1;
MoveL RelTool (p1,40.500000,10.500000,16.425089,\Rx:=0.000000,\Ry:=-0.803938),vel1,zoneval,Extruder\WObj:=Workobject_1;
MoveL RelTool (p1,38.000000,10.500000,16.225576,\Rx:=0.000000,\Ry:=-1.705318),vel1,zoneval,Extruder\WObj:=Workobject_1;
MoveL RelTool (p1,35.500000,10.500000,15.872237,\Rx:=0.000000,\Ry:=-2.219265),vel1,zoneval,Extruder\WObj:=Workobject_1;
MoveL RelTool (p1,33.000000,10.500000,15.358103,\Rx:=0.000000,\Ry:=-3.146417),vel1,zoneval,Extruder\WObj:=Workobject_1;
MoveL RelTool (p1,30.500000,10.500000,14.653673,\Rx:=0.000000,\Ry:=-4.036212),vel1,zoneval,Extruder\WObj:=Workobject_1;
MoveL RelTool (p1,28.000000,10.500000,13.728221,\Rx:=0.000000,\Ry:=-5.244430),vel1,zoneval,Extruder\WObj:=Workobject_1;
MoveL RelTool (p1,25.500000,10.500000,12.502126,\Rx:=0.000000,\Ry:=-6.947078),vel1,zoneval,Extruder\WObj:=Workobject_1;
MoveL RelTool (p1,23.000000,10.500000,10.785467,\Rx:=0.000000,\Ry:=-9.260904),vel1,zoneval,Extruder\WObj:=Workobject_1;
MoveL RelTool (p1,20.500000,10.500000,8.040772,\Rx:=0.000000,\Ry:=-9.245074),vel1,zoneval,Extruder\WObj:=Workobject_1;
MoveL RelTool (p1,18.000000,10.500000,6.640720,\Rx:=0.000000,\Ry:=-2.301628),vel1,zoneval,Extruder\WObj:=Workobject_1;
MoveL RelTool (p1,15.500000,10.500000,6.500000,\Rx:=0.000000,\Ry:=0.000000),vel1,zoneval,Extruder\WObj:=Workobject_1;
MoveL RelTool (p1,13.000000,10.500000,6.500000,\Rx:=0.000000,\Ry:=0.000000),vel1,zoneval,Extruder\WObj:=Workobject_1;
MoveL RelTool (p1,10.500000,10.500000,6.500000,\Rx:=0.000000,\Ry:=0.000000),vel1,zoneval,Extruder\WObj:=Workobject_1;
MoveL RelTool (p1,8.000000,10.500000,6.500000,\Rx:=0.000000,\Ry:=0.000000),vel1,zoneval,Extruder\WObj:=Workobject_1;
MoveL RelTool (p1,5.500000,10.500000,6.500000,\Rx:=0.000000,\Ry:=0.000000),vel1,zoneval,Extruder\WObj:=Workobject_1;
MoveL RelTool (p1,3.000000,10.500000,6.500000,\Rx:=0.000000,\Ry:=0.000000),vel1,zoneval,Extruder\WObj:=Workobject_1;
